LIN {X 0,Y 143.152,Z 440.148,A -85,B 0,C 180,E1 -24453.78,E2 -24453.78} C_VEL
LIN {X 0,Y 143.303,Z 440.124,A -85,B 0,C 180,E1 -24459.924,E2 -24459.924} C_VEL
LIN {X 0,Y 143.35,Z 440.119,A -85,B 0,C 180,E1 -24465.812,E2 -24465.812} C_VEL
LIN {X 0,Y 143.533,Z 440.103,A -85,B 0,C 180,E1 -24468.707,E2 -24468.707} C_VEL
LIN {X 0,Y 143.622,Z 440.089,A -85,B 0,C 180,E1 -24471.56,E2 -24471.56} C_VEL
LIN {X 0,Y 144.173,Z 439.992,A -85,B 0,C 180,E1 -24480.002,E2 -24480.002} C_VEL
LIN {X 0,Y 143.623,Z 440.096,A -85,B 0,C 180,E1 -24488.443,E2 -24488.443} C_VEL
LIN {X 0,Y 143.503,Z 440.112,A -85,B 0,C 180,E1 -24491.63,E2 -24491.63} C_VEL
LIN {X 0,Y 143.297,Z 440.142,A -85,B 0,C 180,E1 -24497.115,E2 -24497.115} C_VEL
LIN {X 0,Y 143.385,Z 440.981,A -85,B 0,C 180,E1 -24501.367,E2 -24501.367} C_VEL
LIN {X 0,Y 143.555,Z 442.59,A -85,B 0,C 180,E1 -24508.212,E2 -24508.212} C_VEL
LIN {X 0,Y 143.628,Z 443.352,A -85,B 0,C 180,E1 -24510.714,E2 -24510.714} C_VEL
LIN {X 0,Y 144.738,Z 446.525,A -85,B 0,C 180,E1 -24511.876,E2 -24511.876} C_VEL
LIN {X 0,Y 147.342,Z 449.815,A -85,B 0,C 180,E1 -24513.997,E2 -24513.997} C_VEL
LIN {X 0,Y 148.899,Z 453.219,A -85,B 0,C 180,E1 -24515.429,E2 -24515.429} C_VEL
LIN {X 0,Y 150.409,Z 455.407,A -85,B 0,C 180,E1 -24516.568,E2 -24516.568} C_VEL
LIN {X 0,Y 153.168,Z 461.405,A -85,B 0,C 180,E1 -24519.035,E2 -24519.035} C_VEL
LIN {X 0,Y 155.875,Z 468.036,A -85,B 0,C 180,E1 -24521.519,E2 -24521.519} C_VEL
LIN {X 0,Y 158.224,Z 476.972,A -85,B 0,C 180,E1 -24524.486,E2 -24524.486} C_VEL
LIN {X 0,Y 159.487,Z 487.574,A -85,B 0,C 180,E1 -24527.779,E2 -24527.779} C_VEL
LIN {X 0,Y 159.695,Z 496.347,A -85,B 0,C 180,E1 -24530.573,E2 -24530.573} C_VEL
LIN {X 0,Y 159.089,Z 505.794,A -85,B 0,C 180,E1 -24533.831,E2 -24533.831} C_VEL
LIN {X 0,Y 158.048,Z 512.286,A -85,B 0,C 180,E1 -24536.232,E2 -24536.232} C_VEL
LIN {X 0,Y 154.375,Z 520.117,A -85,B 0,C 180,E1 -24539.193,E2 -24539.193} C_VEL
LIN {X 0,Y 151.127,Z 526.657,A -85,B 0,C 180,E1 -24542.288,E2 -24542.288} C_VEL
LIN {X 0,Y 148.767,Z 531.159,A -85,B 0,C 180,E1 -24544.839,E2 -24544.839} C_VEL
LIN {X 0,Y 145.71,Z 536.651,A -85,B 0,C 180,E1 -24548.793,E2 -24548.793} C_VEL
LIN {X 0,Y 143.316,Z 540.978,A -85,B 0,C 180,E1 -24552.889,E2 -24552.889} C_VEL
LIN {X 0,Y 142.25,Z 543.351,A -85,B 0,C 180,E1 -24555.698,E2 -24555.698} C_VEL
LIN {X 0,Y 141.418,Z 545.156,A -85,B 0,C 180,E1 -24558.534,E2 -24558.534} C_VEL
LIN {X 0,Y 140.617,Z 547.617,A -85,B 0,C 180,E1 -24564.263,E2 -24564.263} C_VEL
LIN {X 0,Y 140.572,Z 548.37,A -85,B 0,C 180,E1 -24569.356,E2 -24569.356} C_VEL
LIN {X 0,Y 140.49,Z 548.211,A -85,B 0,C 180,E1 -24572.867,E2 -24572.867} C_VEL
LIN {X 0,Y 140.558,Z 547.615,A -85,B 0,C 180,E1 -24575.739,E2 -24575.739} C_VEL
LIN {X 0,Y 141.418,Z 545.156,A -85,B 0,C 180,E1 -24581.466,E2 -24581.466} C_VEL
LIN {X 0,Y 142.745,Z 542.198,A -85,B 0,C 180,E1 -24585.711,E2 -24585.711} C_VEL
LIN {X 0,Y 144.854,Z 538.206,A -85,B 0,C 180,E1 -24589.854,E2 -24589.854} C_VEL
LIN {X 0,Y 147.638,Z 533.074,A -85,B 0,C 180,E1 -24593.867,E2 -24593.867} C_VEL
LIN {X 0,Y 150.526,Z 527.813,A -85,B 0,C 180,E1 -24597.079,E2 -24597.079} C_VEL
LIN {X 0,Y 152.903,Z 523.006,A -85,B 0,C 180,E1 -24599.535,E2 -24599.535} C_VEL
LIN {X 0,Y 155.803,Z 517.169,A -85,B 0,C 180,E1 -24602.006,E2 -24602.006} C_VEL
LIN {X 0,Y 157.995,Z 512.284,A -85,B 0,C 180,E1 -24603.781,E2 -24603.781} C_VEL
LIN {X 0,Y 159.283,Z 504.165,A -85,B 0,C 180,E1 -24606.777,E2 -24606.777} C_VEL
LIN {X 0,Y 159.691,Z 494.189,A -85,B 0,C 180,E1 -24610.136,E2 -24610.136} C_VEL
LIN {X 0,Y 159.209,Z 484.217,A -85,B 0,C 180,E1 -24613.246,E2 -24613.246} C_VEL
LIN {X 0,Y 157.654,Z 474.494,A -85,B 0,C 180,E1 -24616.289,E2 -24616.289} C_VEL
LIN {X 0,Y 155.43,Z 466.702,A -85,B 0,C 180,E1 -24618.95,E2 -24618.95} C_VEL
LIN {X 0,Y 152.654,Z 459.906,A -85,B 0,C 180,E1 -24621.503,E2 -24621.503} C_VEL
LIN {X 0,Y 150.327,Z 455.158,A -85,B 0,C 180,E1 -24623.513,E2 -24623.513} C_VEL
LIN {X 0,Y 147.761,Z 451.088,A -85,B 0,C 180,E1 -24625.549,E2 -24625.549} C_VEL
LIN {X 0,Y 147.026,Z 449.221,A -85,B 0,C 180,E1 -24626.287,E2 -24626.287} C_VEL
LIN {X 0,Y 144.65,Z 446.353,A -85,B 0,C 180,E1 -24628.205,E2 -24628.205} C_VEL
LIN {X 0,Y 143.667,Z 443.599,A -85,B 0,C 180,E1 -24629.193,E2 -24629.193} C_VEL
LIN {X 0,Y 143.581,Z 443.188,A -85,B 0,C 180,E1 -24629.478,E2 -24629.478} C_VEL
LIN {X 0,Y 143.46,Z 442.211,A -85,B 0,C 180,E1 -24633.299,E2 -24633.299} C_VEL
LIN {X 0,Y 142.742,Z 441.762,A -85,B 0,C 180,E1 -24635.632,E2 -24635.632} C_VEL
LIN {X 0,Y 141.111,Z 441.498,A -85,B 0,C 180,E1 -24637.936,E2 -24637.936} C_VEL
LIN {X 0,Y 136.544,Z 441.058,A -85,B 0,C 180,E1 -24644.298,E2 -24644.298} C_VEL
LIN {X 0,Y 136.275,Z 441.006,A -85,B 0,C 180,E1 -24645.981,E2 -24645.981} C_VEL
LIN {X 0,Y 136.549,Z 440.977,A -85,B 0,C 180,E1 -24651.116,E2 -24651.116} C_VEL
LIN {X 0,Y 137.13,Z 440.867,A -85,B 0,C 180,E1 -24659.998,E2 -24659.998} C_VEL
LIN {X 0,Y 136.549,Z 440.967,A -85,B 0,C 180,E1 -24668.881,E2 -24668.881} C_VEL
LIN {X 0,Y 136.437,Z 440.991,A -85,B 0,C 180,E1 -24671.889,E2 -24671.889} C_VEL
LIN {X 0,Y 136.235,Z 441.013,A -85,B 0,C 180,E1 -24678.029,E2 -24678.029} C_VEL
LIN {X 0,Y 136.194,Z 441.018,A -85,B 0,C 180,E1 -24681.747,E2 -24681.747} C_VEL
LIN {X 0,Y 136.08,Z 441.049,A -85,B 0,C 180,E1 -24685.115,E2 -24685.115} C_VEL
LIN {X 0,Y 136.755,Z 443.236,A -85,B 0,C 180,E1 -24686.104,E2 -24686.104} C_VEL
LIN {X 0,Y 138.766,Z 445.73,A -85,B 0,C 180,E1 -24688.327,E2 -24688.327} C_VEL
LIN {X 0,Y 140.093,Z 446.714,A -85,B 0,C 180,E1 -24689.543,E2 -24689.543} C_VEL
LIN {X 0,Y 141.491,Z 449.595,A -85,B 0,C 180,E1 -24691.122,E2 -24691.122} C_VEL
LIN {X 0,Y 143.665,Z 452.032,A -85,B 0,C 180,E1 -24693.012,E2 -24693.012} C_VEL
LIN {X 0,Y 145.332,Z 454.972,A -85,B 0,C 180,E1 -24694.707,E2 -24694.707} C_VEL
LIN {X 0,Y 148.827,Z 460.554,A -85,B 0,C 180,E1 -24697.87,E2 -24697.87} C_VEL
LIN {X 0,Y 153.54,Z 470.176,A -85,B 0,C 180,E1 -24702.464,E2 -24702.464} C_VEL
LIN {X 0,Y 157.143,Z 479.374,A -85,B 0,C 180,E1 -24706.461,E2 -24706.461} C_VEL
LIN {X 0,Y 159.474,Z 487.535,A -85,B 0,C 180,E1 -24709.834,E2 -24709.834} C_VEL
LIN {X 0,Y 161.218,Z 496.736,A -85,B 0,C 180,E1 -24713.624,E2 -24713.624} C_VEL
LIN {X 0,Y 162.342,Z 505.111,A -85,B 0,C 180,E1 -24717.36,E2 -24717.36} C_VEL
LIN {X 0,Y 164.436,Z 512.684,A -85,B 0,C 180,E1 -24721.389,E2 -24721.389} C_VEL
LIN {X 0,Y 167.413,Z 518.734,A -85,B 0,C 180,E1 -24725.179,E2 -24725.179} C_VEL
LIN {X 0,Y 170.704,Z 523.029,A -85,B 0,C 180,E1 -24728.252,E2 -24728.252} C_VEL
LIN {X 0,Y 176.708,Z 528.218,A -85,B 0,C 180,E1 -24732.649,E2 -24732.649} C_VEL
LIN {X 0,Y 183.955,Z 532.227,A -85,B 0,C 180,E1 -24736.749,E2 -24736.749} C_VEL
LIN {X 0,Y 192.338,Z 535.226,A -85,B 0,C 180,E1 -24740.593,E2 -24740.593} C_VEL
LIN {X 0,Y 200.865,Z 537.166,A -85,B 0,C 180,E1 -24743.975,E2 -24743.975} C_VEL
LIN {X 0,Y 206.622,Z 538.036,A -85,B 0,C 180,E1 -24746.099,E2 -24746.099} C_VEL
LIN {X 0,Y 212.047,Z 538.453,A -85,B 0,C 180,E1 -24748.101,E2 -24748.101} C_VEL
LIN {X 0,Y 216.311,Z 538.505,A -85,B 0,C 180,E1 -24750,E2 -24750} C_VEL
LIN {X 0,Y 211.001,Z 538.385,A -85,B 0,C 180,E1 -24752.268,E2 -24752.268} C_VEL
LIN {X 0,Y 204.489,Z 537.779,A -85,B 0,C 180,E1 -24754.678,E2 -24754.678} C_VEL
LIN {X 0,Y 195.02,Z 535.982,A -85,B 0,C 180,E1 -24758.288,E2 -24758.288} C_VEL
LIN {X 0,Y 186.734,Z 533.39,A -85,B 0,C 180,E1 -24761.896,E2 -24761.896} C_VEL
LIN {X 0,Y 178.979,Z 529.663,A -85,B 0,C 180,E1 -24765.954,E2 -24765.954} C_VEL
LIN {X 0,Y 174.564,Z 526.656,A -85,B 0,C 180,E1 -24768.788,E2 -24768.788} C_VEL
LIN {X 0,Y 169.225,Z 521.23,A -85,B 0,C 180,E1 -24773.069,E2 -24773.069} C_VEL
LIN {X 0,Y 165.611,Z 515.406,A -85,B 0,C 180,E1 -24776.982,E2 -24776.982} C_VEL
LIN {X 0,Y 163.318,Z 509.057,A -85,B 0,C 180,E1 -24780.613,E2 -24780.613} C_VEL
LIN {X 0,Y 162.063,Z 503.157,A -85,B 0,C 180,E1 -24783.563,E2 -24783.563} C_VEL
LIN {X 0,Y 160.944,Z 494.761,A -85,B 0,C 180,E1 -24787.167,E2 -24787.167} C_VEL
LIN {X 0,Y 159.114,Z 486.266,A -85,B 0,C 180,E1 -24790.677,E2 -24790.677} C_VEL
LIN {X 0,Y 156.632,Z 477.951,A -85,B 0,C 180,E1 -24794.12,E2 -24794.12} C_VEL
LIN {X 0,Y 152.851,Z 468.714,A -85,B 0,C 180,E1 -24798.189,E2 -24798.189} C_VEL
LIN {X 0,Y 148.798,Z 460.661,A -85,B 0,C 180,E1 -24802.122,E2 -24802.122} C_VEL
LIN {X 0,Y 145.994,Z 455.806,A -85,B 0,C 180,E1 -24804.715,E2 -24804.715} C_VEL
LIN {X 0,Y 143.909,Z 452.642,A -85,B 0,C 180,E1 -24806.707,E2 -24806.707} C_VEL
LIN {X 0,Y 143.083,Z 451.254,A -85,B 0,C 180,E1 -24807.506,E2 -24807.506} C_VEL
LIN {X 0,Y 140.829,Z 448.546,A -85,B 0,C 180,E1 -24809.548,E2 -24809.548} C_VEL
LIN {X 0,Y 139.946,Z 446.499,A -85,B 0,C 180,E1 -24810.611,E2 -24810.611} C_VEL
LIN {X 0,Y 137.323,Z 444.183,A -85,B 0,C 180,E1 -24813.193,E2 -24813.193} C_VEL
LIN {X 0,Y 136.247,Z 441.855,A -85,B 0,C 180,E1 -24814.612,E2 -24814.612} C_VEL
LIN {X 0,Y 136.079,Z 441.024,A -85,B 0,C 180,E1 -24814.987,E2 -24814.987} C_VEL
LIN {X 0,Y 136.239,Z 441.008,A -85,B 0,C 180,E1 -24818.834,E2 -24818.834} C_VEL
LIN {X 0,Y 136.26,Z 441.001,A -85,B 0,C 180,E1 -24825.057,E2 -24825.057} C_VEL
LIN {X 0,Y 136.428,Z 440.991,A -85,B 0,C 180,E1 -24828.167,E2 -24828.167} C_VEL
LIN {X 0,Y 136.548,Z 440.967,A -85,B 0,C 180,E1 -24831.119,E2 -24831.119} C_VEL
LIN {X 0,Y 137.13,Z 440.867,A -85,B 0,C 180,E1 -24840.002,E2 -24840.002} C_VEL
LIN {X 0,Y 136.549,Z 440.976,A -85,B 0,C 180,E1 -24848.884,E2 -24848.884} C_VEL
LIN {X 0,Y 136.439,Z 440.993,A -85,B 0,C 180,E1 -24851.892,E2 -24851.892} C_VEL
LIN {X 0,Y 136.262,Z 441.014,A -85,B 0,C 180,E1 -24854.946,E2 -24854.946} C_VEL
LIN {X 0,Y 136.364,Z 442.037,A -85,B 0,C 180,E1 -24861.149,E2 -24861.149} C_VEL
LIN {X 0,Y 136.444,Z 443.198,A -85,B 0,C 180,E1 -24865.251,E2 -24865.251} C_VEL
LIN {X 0,Y 137.466,Z 445.953,A -85,B 0,C 180,E1 -24866.575,E2 -24866.575} C_VEL
LIN {X 0,Y 139.977,Z 449.017,A -85,B 0,C 180,E1 -24869.142,E2 -24869.142} C_VEL
LIN {X 0,Y 140.494,Z 449.746,A -85,B 0,C 180,E1 -24869.662,E2 -24869.662} C_VEL
LIN {X 0,Y 142.053,Z 453.203,A -85,B 0,C 180,E1 -24871.403,E2 -24871.403} C_VEL
LIN {X 0,Y 143.833,Z 455.627,A -85,B 0,C 180,E1 -24872.972,E2 -24872.972} C_VEL
LIN {X 0,Y 145.746,Z 459.585,A -85,B 0,C 180,E1 -24874.942,E2 -24874.942} C_VEL
LIN {X 0,Y 149.295,Z 467.386,A -85,B 0,C 180,E1 -24878.488,E2 -24878.488} C_VEL
LIN {X 0,Y 151.713,Z 475.064,A -85,B 0,C 180,E1 -24881.511,E2 -24881.511} C_VEL
LIN {X 0,Y 152.981,Z 482.109,A -85,B 0,C 180,E1 -24883.986,E2 -24883.986} C_VEL
LIN {X 0,Y 153.608,Z 490.094,A -85,B 0,C 180,E1 -24886.664,E2 -24886.664} C_VEL
LIN {X 0,Y 153.606,Z 496.767,A -85,B 0,C 180,E1 -24888.922,E2 -24888.922} C_VEL
LIN {X 0,Y 153.015,Z 505.059,A -85,B 0,C 180,E1 -24891.926,E2 -24891.926} C_VEL
LIN {X 0,Y 151.949,Z 512.081,A -85,B 0,C 180,E1 -24894.68,E2 -24894.68} C_VEL
LIN {X 0,Y 150.668,Z 515.347,A -85,B 0,C 180,E1 -24895.963,E2 -24895.963} C_VEL
LIN {X 0,Y 147.535,Z 521.295,A -85,B 0,C 180,E1 -24898.4,E2 -24898.4} C_VEL
LIN {X 0,Y 144.83,Z 526.459,A -85,B 0,C 180,E1 -24900.971,E2 -24900.971} C_VEL
LIN {X 0,Y 142.372,Z 530.962,A -85,B 0,C 180,E1 -24903.624,E2 -24903.624} C_VEL
LIN {X 0,Y 139.088,Z 536.453,A -85,B 0,C 180,E1 -24907.731,E2 -24907.731} C_VEL
LIN {X 0,Y 136.51,Z 540.78,A -85,B 0,C 180,E1 -24912.007,E2 -24912.007} C_VEL
LIN {X 0,Y 135.352,Z 543.153,A -85,B 0,C 180,E1 -24914.953,E2 -24914.953} C_VEL
LIN {X 0,Y 134.452,Z 544.958,A -85,B 0,C 180,E1 -24917.932,E2 -24917.932} C_VEL
LIN {X 0,Y 133.543,Z 547.419,A -85,B 0,C 180,E1 -24923.958,E2 -24923.958} C_VEL
LIN {X 0,Y 133.414,Z 548.014,A -85,B 0,C 180,E1 -24926.98,E2 -24926.98} C_VEL
LIN {X 0,Y 133.536,Z 548.175,A -85,B 0,C 180,E1 -24930,E2 -24930} C_VEL
LIN {X 0,Y 133.401,Z 548.014,A -85,B 0,C 180,E1 -24933.02,E2 -24933.02} C_VEL
LIN {X 0,Y 133.474,Z 547.417,A -85,B 0,C 180,E1 -24936.045,E2 -24936.045} C_VEL
LIN {X 0,Y 134.452,Z 544.958,A -85,B 0,C 180,E1 -24942.068,E2 -24942.068} C_VEL
LIN {X 0,Y 135.884,Z 542,A -85,B 0,C 180,E1 -24946.526,E2 -24946.526} C_VEL
LIN {X 0,Y 138.16,Z 538.008,A -85,B 0,C 180,E1 -24950.859,E2 -24950.859} C_VEL
LIN {X 0,Y 141.152,Z 532.876,A -85,B 0,C 180,E1 -24955.037,E2 -24955.037} C_VEL
LIN {X 0,Y 143.618,Z 528.772,A -85,B 0,C 180,E1 -24957.702,E2 -24957.702} C_VEL
LIN {X 0,Y 146.723,Z 522.808,A -85,B 0,C 180,E1 -24960.912,E2 -24960.912} C_VEL
LIN {X 0,Y 149.807,Z 516.971,A -85,B 0,C 180,E1 -24963.451,E2 -24963.451} C_VEL
LIN {X 0,Y 151.364,Z 513.716,A -85,B 0,C 180,E1 -24964.664,E2 -24964.664} C_VEL
LIN {X 0,Y 152.584,Z 508.373,A -85,B 0,C 180,E1 -24966.782,E2 -24966.782} C_VEL
LIN {X 0,Y 153.37,Z 501.695,A -85,B 0,C 180,E1 -24969.313,E2 -24969.313} C_VEL
LIN {X 0,Y 153.667,Z 493.139,A -85,B 0,C 180,E1 -24972.324,E2 -24972.324} C_VEL
LIN {X 0,Y 153.368,Z 485.551,A -85,B 0,C 180,E1 -24974.895,E2 -24974.895} C_VEL
LIN {X 0,Y 152.082,Z 476.72,A -85,B 0,C 180,E1 -24977.924,E2 -24977.924} C_VEL
LIN {X 0,Y 149.999,Z 469.293,A -85,B 0,C 180,E1 -24980.692,E2 -24980.692} C_VEL
LIN {X 0,Y 147.381,Z 463.041,A -85,B 0,C 180,E1 -24983.409,E2 -24983.409} C_VEL
LIN {X 0,Y 145.755,Z 459.586,A -85,B 0,C 180,E1 -24985.053,E2 -24985.053} C_VEL
LIN {X 0,Y 143.834,Z 455.622,A -85,B 0,C 180,E1 -24987.028,E2 -24987.028} C_VEL
LIN {X 0,Y 140.918,Z 451.084,A -85,B 0,C 180,E1 -24989.773,E2 -24989.773} C_VEL
LIN {X 0,Y 140.363,Z 449.264,A -85,B 0,C 180,E1 -24990.53,E2 -24990.53} C_VEL
LIN {X 0,Y 137.692,Z 446.36,A -85,B 0,C 180,E1 -24993.165,E2 -24993.165} C_VEL
LIN {X 0,Y 136.48,Z 443.495,A -85,B 0,C 180,E1 -24994.654,E2 -24994.654} C_VEL
LIN {X 0,Y 136.387,Z 442.867,A -85,B 0,C 180,E1 -24994.942,E2 -24994.942} C_VEL
LIN {X 0,Y 136.363,Z 442.035,A -85,B 0,C 180,E1 -24998.851,E2 -24998.851} C_VEL
LIN {X 0,Y 136.262,Z 441.012,A -85,B 0,C 180,E1 -25005.054,E2 -25005.054} C_VEL
LIN {X 0,Y 136.275,Z 441.006,A -85,B 0,C 180,E1 -25005.981,E2 -25005.981} C_VEL
LIN {X 0,Y 135.666,Z 441.087,A -85,B 0,C 180,E1 -25008.449,E2 -25008.449} C_VEL
LIN {X 0,Y 134.131,Z 441.278,A -85,B 0,C 180,E1 -25010.888,E2 -25010.888} C_VEL
LIN {X 0,Y 130.654,Z 441.709,A -85,B 0,C 180,E1 -25015.879,E2 -25015.879} C_VEL
LIN {X 0,Y 129.914,Z 441.783,A -85,B 0,C 180,E1 -25018.501,E2 -25018.501} C_VEL
LIN {X 0,Y 129.972,Z 441.761,A -85,B 0,C 180,E1 -25019.384,E2 -25019.384} C_VEL
LIN {X 0,Y 130.085,Z 441.743,A -85,B 0,C 180,E1 -25019.998,E2 -25019.998} C_VEL
LIN {X 0,Y 129.472,Z 441.847,A -85,B 0,C 180,E1 -25029.37,E2 -25029.37} C_VEL
LIN {X 0,Y 129.341,Z 441.874,A -85,B 0,C 180,E1 -25032.552,E2 -25032.552} C_VEL
LIN {X 0,Y 129.192,Z 442.042,A -85,B 0,C 180,E1 -25037.612,E2 -25037.612} C_VEL
LIN {X 0,Y 129.975,Z 444.408,A -85,B 0,C 180,E1 -25039.339,E2 -25039.339} C_VEL
LIN {X 0,Y 132.566,Z 447.181,A -85,B 0,C 180,E1 -25043.163,E2 -25043.163} C_VEL
LIN {X 0,Y 133.355,Z 447.728,A -85,B 0,C 180,E1 -25044.105,E2 -25044.105} C_VEL
LIN {X 0,Y 134.792,Z 450.708,A -85,B 0,C 180,E1 -25046.201,E2 -25046.201} C_VEL
LIN {X 0,Y 137.341,Z 453.815,A -85,B 0,C 180,E1 -25049.087,E2 -25049.087} C_VEL
LIN {X 0,Y 138.451,Z 455.857,A -85,B 0,C 180,E1 -25050.503,E2 -25050.503} C_VEL
LIN {X 0,Y 139.798,Z 457.375,A -85,B 0,C 180,E1 -25051.859,E2 -25051.859} C_VEL
LIN {X 0,Y 143.013,Z 463.032,A -85,B 0,C 180,E1 -25055.353,E2 -25055.353} C_VEL
LIN {X 0,Y 146.78,Z 470.562,A -85,B 0,C 180,E1 -25059.522,E2 -25059.522} C_VEL
LIN {X 0,Y 150.046,Z 478.638,A -85,B 0,C 180,E1 -25063.518,E2 -25063.518} C_VEL
LIN {X 0,Y 152.68,Z 487.147,A -85,B 0,C 180,E1 -25067.431,E2 -25067.431} C_VEL
LIN {X 0,Y 154.244,Z 494.584,A -85,B 0,C 180,E1 -25070.766,E2 -25070.766} C_VEL
LIN {X 0,Y 155.145,Z 501.503,A -85,B 0,C 180,E1 -25073.922,E2 -25073.922} C_VEL
LIN {X 0,Y 156.187,Z 509.493,A -85,B 0,C 180,E1 -25077.924,E2 -25077.924} C_VEL
LIN {X 0,Y 158.536,Z 516.995,A -85,B 0,C 180,E1 -25082.448,E2 -25082.448} C_VEL
LIN {X 0,Y 162.311,Z 523.278,A -85,B 0,C 180,E1 -25087.065,E2 -25087.065} C_VEL
LIN {X 0,Y 167.764,Z 528.419,A -85,B 0,C 180,E1 -25091.646,E2 -25091.646} C_VEL
LIN {X 0,Y 174.661,Z 532.488,A -85,B 0,C 180,E1 -25096.03,E2 -25096.03} C_VEL
LIN {X 0,Y 179.811,Z 534.632,A -85,B 0,C 180,E1 -25098.731,E2 -25098.731} C_VEL
LIN {X 0,Y 185.399,Z 536.246,A -85,B 0,C 180,E1 -25101.279,E2 -25101.279} C_VEL
LIN {X 0,Y 197.271,Z 538.308,A -85,B 0,C 180,E1 -25105.955,E2 -25105.955} C_VEL
LIN {X 0,Y 203.89,Z 538.764,A -85,B 0,C 180,E1 -25108.373,E2 -25108.373} C_VEL
LIN {X 0,Y 207.943,Z 538.733,A -85,B 0,C 180,E1 -25110,E2 -25110} C_VEL
LIN {X 0,Y 202.902,Z 538.706,A -85,B 0,C 180,E1 -25111.985,E2 -25111.985} C_VEL
LIN {X 0,Y 197.148,Z 538.298,A -85,B 0,C 180,E1 -25114.088,E2 -25114.088} C_VEL
LIN {X 0,Y 184.954,Z 536.128,A -85,B 0,C 180,E1 -25118.906,E2 -25118.906} C_VEL
LIN {X 0,Y 179.306,Z 534.463,A -85,B 0,C 180,E1 -25121.518,E2 -25121.518} C_VEL
LIN {X 0,Y 172.174,Z 531.319,A -85,B 0,C 180,E1 -25125.401,E2 -25125.401} C_VEL
LIN {X 0,Y 165.053,Z 526.107,A -85,B 0,C 180,E1 -25130.489,E2 -25130.489} C_VEL
LIN {X 0,Y 160.65,Z 520.863,A -85,B 0,C 180,E1 -25134.757,E2 -25134.757} C_VEL
LIN {X 0,Y 157.739,Z 515.011,A -85,B 0,C 180,E1 -25138.792,E2 -25138.792} C_VEL
LIN {X 0,Y 155.969,Z 508.24,A -85,B 0,C 180,E1 -25142.732,E2 -25142.732} C_VEL
LIN {X 0,Y 155.167,Z 501.502,A -85,B 0,C 180,E1 -25146.072,E2 -25146.072} C_VEL
LIN {X 0,Y 154.242,Z 494.588,A -85,B 0,C 180,E1 -25149.234,E2 -25149.234} C_VEL
LIN {X 0,Y 152.679,Z 487.149,A -85,B 0,C 180,E1 -25152.568,E2 -25152.568} C_VEL
LIN {X 0,Y 150.029,Z 478.61,A -85,B 0,C 180,E1 -25156.498,E2 -25156.498} C_VEL
LIN {X 0,Y 146.751,Z 470.581,A -85,B 0,C 180,E1 -25160.486,E2 -25160.486} C_VEL
LIN {X 0,Y 142.215,Z 461.47,A -85,B 0,C 180,E1 -25165.551,E2 -25165.551} C_VEL
LIN {X 0,Y 140.368,Z 458.597,A -85,B 0,C 180,E1 -25167.438,E2 -25167.438} C_VEL
LIN {X 0,Y 139.797,Z 457.38,A -85,B 0,C 180,E1 -25168.141,E2 -25168.141} C_VEL
LIN {X 0,Y 138.121,Z 455.345,A -85,B 0,C 180,E1 -25169.882,E2 -25169.882} C_VEL
LIN {X 0,Y 136.142,Z 452.123,A -85,B 0,C 180,E1 -25172.317,E2 -25172.317} C_VEL
LIN {X 0,Y 133.974,Z 449.353,A -85,B 0,C 180,E1 -25174.878,E2 -25174.878} C_VEL
LIN {X 0,Y 133.227,Z 447.52,A -85,B 0,C 180,E1 -25176.077,E2 -25176.077} C_VEL
LIN {X 0,Y 130.715,Z 445.463,A -85,B 0,C 180,E1 -25179.397,E2 -25179.397} C_VEL
LIN {X 0,Y 129.515,Z 443.301,A -85,B 0,C 180,E1 -25181.616,E2 -25181.616} C_VEL
LIN {X 0,Y 129.19,Z 441.893,A -85,B 0,C 180,E1 -25182.592,E2 -25182.592} C_VEL
LIN {X 0,Y 129.373,Z 441.87,A -85,B 0,C 180,E1 -25187.905,E2 -25187.905} C_VEL
LIN {X 0,Y 129.471,Z 441.847,A -85,B 0,C 180,E1 -25190.63,E2 -25190.63} C_VEL
LIN {X 0,Y 130.085,Z 441.743,A -85,B 0,C 180,E1 -25200.002,E2 -25200.002} C_VEL
LIN {X 0,Y 129.472,Z 441.858,A -85,B 0,C 180,E1 -25209.374,E2 -25209.374} C_VEL
LIN {X 0,Y 129.342,Z 441.876,A -85,B 0,C 180,E1 -25212.555,E2 -25212.555} C_VEL
LIN {X 0,Y 129.261,Z 442.629,A -85,B 0,C 180,E1 -25217.3,E2 -25217.3} C_VEL
LIN {X 0,Y 130.424,Z 445.76,A -85,B 0,C 180,E1 -25219.58,E2 -25219.58} C_VEL
LIN {X 0,Y 133.372,Z 449.115,A -85,B 0,C 180,E1 -25223.692,E2 -25223.692} C_VEL
LIN {X 0,Y 133.814,Z 449.957,A -85,B 0,C 180,E1 -25224.33,E2 -25224.33} C_VEL
LIN {X 0,Y 135.361,Z 453.257,A -85,B 0,C 180,E1 -25226.501,E2 -25226.501} C_VEL
LIN {X 0,Y 137.281,Z 455.719,A -85,B 0,C 180,E1 -25228.579,E2 -25228.579} C_VEL
LIN {X 0,Y 138.82,Z 459.231,A -85,B 0,C 180,E1 -25230.612,E2 -25230.612} C_VEL
LIN {X 0,Y 139.967,Z 460.897,A -85,B 0,C 180,E1 -25231.818,E2 -25231.818} C_VEL
LIN {X 0,Y 143.496,Z 468.921,A -85,B 0,C 180,E1 -25235.997,E2 -25235.997} C_VEL
LIN {X 0,Y 145.958,Z 476.275,A -85,B 0,C 180,E1 -25239.287,E2 -25239.287} C_VEL
LIN {X 0,Y 147.347,Z 484.091,A -85,B 0,C 180,E1 -25242.349,E2 -25242.349} C_VEL
LIN {X 0,Y 147.789,Z 492.75,A -85,B 0,C 180,E1 -25245.507,E2 -25245.507} C_VEL
LIN {X 0,Y 147.255,Z 503.201,A -85,B 0,C 180,E1 -25249.404,E2 -25249.404} C_VEL
LIN {X 0,Y 145.888,Z 511.872,A -85,B 0,C 180,E1 -25252.975,E2 -25252.975} C_VEL
LIN {X 0,Y 144.799,Z 515.148,A -85,B 0,C 180,E1 -25254.379,E2 -25254.379} C_VEL
LIN {X 0,Y 141.515,Z 521.097,A -85,B 0,C 180,E1 -25256.888,E2 -25256.888} C_VEL
LIN {X 0,Y 137.991,Z 527.352,A -85,B 0,C 180,E1 -25260.18,E2 -25260.18} C_VEL
LIN {X 0,Y 136.047,Z 530.765,A -85,B 0,C 180,E1 -25262.295,E2 -25262.295} C_VEL
LIN {X 0,Y 132.519,Z 536.255,A -85,B 0,C 180,E1 -25266.563,E2 -25266.563} C_VEL
LIN {X 0,Y 129.742,Z 540.581,A -85,B 0,C 180,E1 -25271.034,E2 -25271.034} C_VEL
LIN {X 0,Y 128.466,Z 542.955,A -85,B 0,C 180,E1 -25274.126,E2 -25274.126} C_VEL
LIN {X 0,Y 127.481,Z 544.76,A -85,B 0,C 180,E1 -25277.261,E2 -25277.261} C_VEL
LIN {X 0,Y 126.464,Z 547.222,A -85,B 0,C 180,E1 -25283.619,E2 -25283.619} C_VEL
LIN {X 0,Y 126.317,Z 547.817,A -85,B 0,C 180,E1 -25286.811,E2 -25286.811} C_VEL
LIN {X 0,Y 126.432,Z 547.978,A -85,B 0,C 180,E1 -25290,E2 -25290} C_VEL
LIN {X 0,Y 126.306,Z 547.817,A -85,B 0,C 180,E1 -25293.19,E2 -25293.19} C_VEL
LIN {X 0,Y 126.415,Z 547.22,A -85,B 0,C 180,E1 -25296.384,E2 -25296.384} C_VEL
LIN {X 0,Y 127.481,Z 544.76,A -85,B 0,C 180,E1 -25302.739,E2 -25302.739} C_VEL
LIN {X 0,Y 129.062,Z 541.802,A -85,B 0,C 180,E1 -25307.427,E2 -25307.427} C_VEL
LIN {X 0,Y 131.521,Z 537.81,A -85,B 0,C 180,E1 -25311.965,E2 -25311.965} C_VEL
LIN {X 0,Y 134.739,Z 532.679,A -85,B 0,C 180,E1 -25316.318,E2 -25316.318} C_VEL
LIN {X 0,Y 137.24,Z 528.729,A -85,B 0,C 180,E1 -25318.997,E2 -25318.997} C_VEL
LIN {X 0,Y 140.724,Z 522.472,A -85,B 0,C 180,E1 -25322.47,E2 -25322.47} C_VEL
LIN {X 0,Y 143.923,Z 516.774,A -85,B 0,C 180,E1 -25325.013,E2 -25325.013} C_VEL
LIN {X 0,Y 145.41,Z 513.513,A -85,B 0,C 180,E1 -25326.303,E2 -25326.303} C_VEL
LIN {X 0,Y 146.691,Z 507.118,A -85,B 0,C 180,E1 -25328.995,E2 -25328.995} C_VEL
LIN {X 0,Y 147.49,Z 499.878,A -85,B 0,C 180,E1 -25331.843,E2 -25331.843} C_VEL
LIN {X 0,Y 147.766,Z 491.738,A -85,B 0,C 180,E1 -25334.854,E2 -25334.854} C_VEL
LIN {X 0,Y 147.176,Z 483.046,A -85,B 0,C 180,E1 -25338.044,E2 -25338.044} C_VEL
LIN {X 0,Y 145.656,Z 475.203,A -85,B 0,C 180,E1 -25341.15,E2 -25341.15} C_VEL
LIN {X 0,Y 143.223,Z 468.266,A -85,B 0,C 180,E1 -25344.342,E2 -25344.342} C_VEL
LIN {X 0,Y 139.967,Z 460.897,A -85,B 0,C 180,E1 -25348.182,E2 -25348.182} C_VEL
LIN {X 0,Y 138.11,Z 457.89,A -85,B 0,C 180,E1 -25350.253,E2 -25350.253} C_VEL
LIN {X 0,Y 136.907,Z 455.025,A -85,B 0,C 180,E1 -25351.858,E2 -25351.858} C_VEL
LIN {X 0,Y 134.509,Z 451.848,A -85,B 0,C 180,E1 -25354.567,E2 -25354.567} C_VEL
LIN {X 0,Y 133.549,Z 449.128,A -85,B 0,C 180,E1 -25356.135,E2 -25356.135} C_VEL
LIN {X 0,Y 130.828,Z 446.386,A -85,B 0,C 180,E1 -25359.766,E2 -25359.766} C_VEL
LIN {X 0,Y 129.548,Z 443.693,A -85,B 0,C 180,E1 -25362.027,E2 -25362.027} C_VEL
LIN {X 0,Y 129.228,Z 442.439,A -85,B 0,C 180,E1 -25362.798,E2 -25362.798} C_VEL
LIN {X 0,Y 129.374,Z 441.87,A -85,B 0,C 180,E1 -25367.902,E2 -25367.902} C_VEL
LIN {X 0,Y 129.472,Z 441.858,A -85,B 0,C 180,E1 -25370.626,E2 -25370.626} C_VEL
LIN {X 0,Y 129.972,Z 441.761,A -85,B 0,C 180,E1 -25379.384,E2 -25379.384} C_VEL
LIN {X 0,Y 129.903,Z 441.912,A -85,B 0,C 180,E1 -25381.102,E2 -25381.102} C_VEL
LIN {X 0,Y 128.827,Z 442.724,A -85,B 0,C 180,E1 -25383.643,E2 -25383.643} C_VEL
LIN {X 0,Y 125.305,Z 445.94,A -85,B 0,C 180,E1 -25389.61,E2 -25389.61} C_VEL
LIN {X 0,Y 124.974,Z 447.305,A -85,B 0,C 180,E1 -25392.287,E2 -25392.287} C_VEL
LIN {X 0,Y 125.216,Z 447.687,A -85,B 0,C 180,E1 -25393.181,E2 -25393.181} C_VEL
LIN {X 0,Y 126.971,Z 448.884,A -85,B 0,C 180,E1 -25396.788,E2 -25396.788} C_VEL
LIN {X 0,Y 127.806,Z 451.163,A -85,B 0,C 180,E1 -25398.846,E2 -25398.846} C_VEL
LIN {X 0,Y 130.676,Z 454.297,A -85,B 0,C 180,E1 -25403.323,E2 -25403.323} C_VEL
LIN {X 0,Y 131.731,Z 456.709,A -85,B 0,C 180,E1 -25405.263,E2 -25405.263} C_VEL
LIN {X 0,Y 133.934,Z 459.653,A -85,B 0,C 180,E1 -25408.179,E2 -25408.179} C_VEL
LIN {X 0,Y 135.124,Z 461.883,A -85,B 0,C 180,E1 -25409.797,E2 -25409.797} C_VEL
LIN {X 0,Y 136.223,Z 463.251,A -85,B 0,C 180,E1 -25411.057,E2 -25411.057} C_VEL
LIN {X 0,Y 140.118,Z 470.912,A -85,B 0,C 180,E1 -25416.109,E2 -25416.109} C_VEL
LIN {X 0,Y 143.362,Z 478.793,A -85,B 0,C 180,E1 -25420.586,E2 -25420.586} C_VEL
LIN {X 0,Y 145.712,Z 486.1,A -85,B 0,C 180,E1 -25424.372,E2 -25424.372} C_VEL
LIN {X 0,Y 147.526,Z 493.778,A -85,B 0,C 180,E1 -25428.169,E2 -25428.169} C_VEL
LIN {X 0,Y 148.488,Z 500.347,A -85,B 0,C 180,E1 -25431.389,E2 -25431.389} C_VEL
LIN {X 0,Y 148.994,Z 507.266,A -85,B 0,C 180,E1 -25434.901,E2 -25434.901} C_VEL
LIN {X 0,Y 149.869,Z 513.33,A -85,B 0,C 180,E1 -25438.411,E2 -25438.411} C_VEL
LIN {X 0,Y 151.782,Z 519.211,A -85,B 0,C 180,E1 -25442.418,E2 -25442.418} C_VEL
LIN {X 0,Y 154.175,Z 523.521,A -85,B 0,C 180,E1 -25445.779,E2 -25445.779} C_VEL
LIN {X 0,Y 159.241,Z 528.868,A -85,B 0,C 180,E1 -25450.806,E2 -25450.806} C_VEL
LIN {X 0,Y 165.393,Z 532.748,A -85,B 0,C 180,E1 -25455.229,E2 -25455.229} C_VEL
LIN {X 0,Y 171.882,Z 535.382,A -85,B 0,C 180,E1 -25458.902,E2 -25458.902} C_VEL
LIN {X 0,Y 177.591,Z 536.978,A -85,B 0,C 180,E1 -25461.621,E2 -25461.621} C_VEL
LIN {X 0,Y 187.526,Z 538.563,A -85,B 0,C 180,E1 -25465.701,E2 -25465.701} C_VEL
LIN {X 0,Y 196.804,Z 539.034,A -85,B 0,C 180,E1 -25469.089,E2 -25469.089} C_VEL
LIN {X 0,Y 199.217,Z 538.97,A -85,B 0,C 180,E1 -25470,E2 -25470} C_VEL
LIN {X 0,Y 193.549,Z 538.964,A -85,B 0,C 180,E1 -25472.081,E2 -25472.081} C_VEL
LIN {X 0,Y 183.663,Z 538.054,A -85,B 0,C 180,E1 -25475.798,E2 -25475.798} C_VEL
LIN {X 0,Y 175.773,Z 536.512,A -85,B 0,C 180,E1 -25479.203,E2 -25479.203} C_VEL
LIN {X 0,Y 170.374,Z 534.899,A -85,B 0,C 180,E1 -25481.903,E2 -25481.903} C_VEL
LIN {X 0,Y 161.842,Z 530.737,A -85,B 0,C 180,E1 -25487.192,E2 -25487.192} C_VEL
LIN {X 0,Y 157.335,Z 527.157,A -85,B 0,C 180,E1 -25490.937,E2 -25490.937} C_VEL
LIN {X 0,Y 152.937,Z 521.428,A -85,B 0,C 180,E1 -25495.882,E2 -25495.882} C_VEL
LIN {X 0,Y 150.5,Z 515.567,A -85,B 0,C 180,E1 -25500.131,E2 -25500.131} C_VEL
LIN {X 0,Y 149.284,Z 509.768,A -85,B 0,C 180,E1 -25503.728,E2 -25503.728} C_VEL
LIN {X 0,Y 148.645,Z 501.728,A -85,B 0,C 180,E1 -25507.925,E2 -25507.925} C_VEL
LIN {X 0,Y 147.693,Z 494.961,A -85,B 0,C 180,E1 -25511.285,E2 -25511.285} C_VEL
LIN {X 0,Y 146.175,Z 487.728,A -85,B 0,C 180,E1 -25514.836,E2 -25514.836} C_VEL
LIN {X 0,Y 143.966,Z 480.609,A -85,B 0,C 180,E1 -25518.505,E2 -25518.505} C_VEL
LIN {X 0,Y 140.635,Z 472.229,A -85,B 0,C 180,E1 -25523.155,E2 -25523.155} C_VEL
LIN {X 0,Y 137.801,Z 466.425,A -85,B 0,C 180,E1 -25526.754,E2 -25526.754} C_VEL
LIN {X 0,Y 136.218,Z 463.262,A -85,B 0,C 180,E1 -25528.942,E2 -25528.942} C_VEL
LIN {X 0,Y 134.501,Z 460.821,A -85,B 0,C 180,E1 -25531.004,E2 -25531.004} C_VEL
LIN {X 0,Y 132.822,Z 458.076,A -85,B 0,C 180,E1 -25533.274,E2 -25533.274} C_VEL
LIN {X 0,Y 131.226,Z 455.762,A -85,B 0,C 180,E1 -25535.566,E2 -25535.566} C_VEL
LIN {X 0,Y 130.677,Z 454.293,A -85,B 0,C 180,E1 -25536.677,E2 -25536.677} C_VEL
LIN {X 0,Y 127.522,Z 450.633,A -85,B 0,C 180,E1 -25541.735,E2 -25541.735} C_VEL
LIN {X 0,Y 126.857,Z 448.592,A -85,B 0,C 180,E1 -25543.507,E2 -25543.507} C_VEL
LIN {X 0,Y 123.057,Z 443.72,A -85,B 0,C 180,E1 -25558.775,E2 -25558.775} C_VEL
LIN {X 0,Y 123.112,Z 443.339,A -85,B 0,C 180,E1 -25560.206,E2 -25560.206} C_VEL
LIN {X 0,Y 127.11,Z 449.288,A -85,B 0,C 180,E1 -25576.36,E2 -25576.36} C_VEL
LIN {X 0,Y 128.099,Z 452.236,A -85,B 0,C 180,E1 -25578.805,E2 -25578.805} C_VEL
LIN {X 0,Y 130.261,Z 455.033,A -85,B 0,C 180,E1 -25582.191,E2 -25582.191} C_VEL
LIN {X 0,Y 133.11,Z 460.458,A -85,B 0,C 180,E1 -25586.668,E2 -25586.668} C_VEL
LIN {X 0,Y 133.693,Z 461.216,A -85,B 0,C 180,E1 -25587.387,E2 -25587.387} C_VEL
LIN {X 0,Y 136.329,Z 466.864,A -85,B 0,C 180,E1 -25591.034,E2 -25591.034} C_VEL
LIN {X 0,Y 139.438,Z 475.064,A -85,B 0,C 180,E1 -25595.603,E2 -25595.603} C_VEL
LIN {X 0,Y 141.022,Z 481.153,A -85,B 0,C 180,E1 -25598.534,E2 -25598.534} C_VEL
LIN {X 0,Y 141.868,Z 487.59,A -85,B 0,C 180,E1 -25601.215,E2 -25601.215} C_VEL
LIN {X 0,Y 141.946,Z 495.76,A -85,B 0,C 180,E1 -25604.432,E2 -25604.432} C_VEL
LIN {X 0,Y 141.02,Z 505.404,A -85,B 0,C 180,E1 -25608.381,E2 -25608.381} C_VEL
LIN {X 0,Y 139.495,Z 513.307,A -85,B 0,C 180,E1 -25611.891,E2 -25611.891} C_VEL
LIN {X 0,Y 138.198,Z 516.578,A -85,B 0,C 180,E1 -25613.307,E2 -25613.307} C_VEL
LIN {X 0,Y 133.237,Z 524.905,A -85,B 0,C 180,E1 -25617.272,E2 -25617.272} C_VEL
LIN {X 0,Y 129.777,Z 530.568,A -85,B 0,C 180,E1 -25620.832,E2 -25620.832} C_VEL
LIN {X 0,Y 126.012,Z 536.058,A -85,B 0,C 180,E1 -25625.274,E2 -25625.274} C_VEL
LIN {X 0,Y 123.022,Z 540.384,A -85,B 0,C 180,E1 -25629.955,E2 -25629.955} C_VEL
LIN {X 0,Y 121.621,Z 542.757,A -85,B 0,C 180,E1 -25633.206,E2 -25633.206} C_VEL
LIN {X 0,Y 120.539,Z 544.563,A -85,B 0,C 180,E1 -25636.514,E2 -25636.514} C_VEL
LIN {X 0,Y 119.411,Z 547.025,A -85,B 0,C 180,E1 -25643.24,E2 -25643.24} C_VEL
LIN {X 0,Y 119.231,Z 547.62,A -85,B 0,C 180,E1 -25646.621,E2 -25646.621} C_VEL
LIN {X 0,Y 119.337,Z 547.781,A -85,B 0,C 180,E1 -25650,E2 -25650} C_VEL
LIN {X 0,Y 119.222,Z 547.62,A -85,B 0,C 180,E1 -25653.379,E2 -25653.379} C_VEL
LIN {X 0,Y 119.338,Z 547.022,A -85,B 0,C 180,E1 -25656.764,E2 -25656.764} C_VEL
LIN {X 0,Y 120.539,Z 544.563,A -85,B 0,C 180,E1 -25663.486,E2 -25663.486} C_VEL
LIN {X 0,Y 122.259,Z 541.603,A -85,B 0,C 180,E1 -25668.431,E2 -25668.431} C_VEL
LIN {X 0,Y 124.943,Z 537.612,A -85,B 0,C 180,E1 -25673.187,E2 -25673.187} C_VEL
LIN {X 0,Y 128.405,Z 532.482,A -85,B 0,C 180,E1 -25677.724,E2 -25677.724} C_VEL
LIN {X 0,Y 131.318,Z 527.969,A -85,B 0,C 180,E1 -25680.87,E2 -25680.87} C_VEL
LIN {X 0,Y 134.746,Z 522.274,A -85,B 0,C 180,E1 -25684.103,E2 -25684.103} C_VEL
LIN {X 0,Y 138.148,Z 516.576,A -85,B 0,C 180,E1 -25686.708,E2 -25686.708} C_VEL
LIN {X 0,Y 139.463,Z 513.306,A -85,B 0,C 180,E1 -25688.119,E2 -25688.119} C_VEL
LIN {X 0,Y 141.017,Z 505.408,A -85,B 0,C 180,E1 -25691.618,E2 -25691.618} C_VEL
LIN {X 0,Y 141.829,Z 497.363,A -85,B 0,C 180,E1 -25694.915,E2 -25694.915} C_VEL
LIN {X 0,Y 141.913,Z 490.576,A -85,B 0,C 180,E1 -25697.61,E2 -25697.61} C_VEL
LIN {X 0,Y 141.663,Z 485.051,A -85,B 0,C 180,E1 -25699.837,E2 -25699.837} C_VEL
LIN {X 0,Y 140.258,Z 477.8,A -85,B 0,C 180,E1 -25703.036,E2 -25703.036} C_VEL
LIN {X 0,Y 137.812,Z 470.6,A -85,B 0,C 180,E1 -25706.753,E2 -25706.753} C_VEL
LIN {X 0,Y 135.765,Z 465.746,A -85,B 0,C 180,E1 -25709.705,E2 -25709.705} C_VEL
LIN {X 0,Y 133.695,Z 461.209,A -85,B 0,C 180,E1 -25712.613,E2 -25712.613} C_VEL
LIN {X 0,Y 131.571,Z 457.924,A -85,B 0,C 180,E1 -25715.543,E2 -25715.543} C_VEL
LIN {X 0,Y 130.127,Z 454.888,A -85,B 0,C 180,E1 -25717.993,E2 -25717.993} C_VEL
LIN {X 0,Y 127.586,Z 451.146,A -85,B 0,C 180,E1 -25722.259,E2 -25722.259} C_VEL
LIN {X 0,Y 126.988,Z 449.013,A -85,B 0,C 180,E1 -25723.934,E2 -25723.934} C_VEL
LIN {X 0,Y 123.081,Z 443.541,A -85,B 0,C 180,E1 -25739.385,E2 -25739.385} C_VEL
LIN {X 0,Y 123.121,Z 443.219,A -85,B 0,C 180,E1 -25739.998,E2 -25739.998} C_VEL
LIN {X 0,Y 125.216,Z 447.687,A -85,B 0,C 180,E1 -25753.181,E2 -25753.181} C_VEL
LIN {X 0,Y 125.747,Z 449.133,A -85,B 0,C 180,E1 -25754.84,E2 -25754.84} C_VEL
LIN {X 0,Y 126.053,Z 453.382,A -85,B 0,C 180,E1 -25757.206,E2 -25757.206} C_VEL
LIN {X 0,Y 126.165,Z 457.869,A -85,B 0,C 180,E1 -25759.555,E2 -25759.555} C_VEL
LIN {X 0,Y 126.77,Z 459.669,A -85,B 0,C 180,E1 -25761.164,E2 -25761.164} C_VEL
LIN {X 0,Y 127.688,Z 460.707,A -85,B 0,C 180,E1 -25762.659,E2 -25762.659} C_VEL
LIN {X 0,Y 129.404,Z 463.97,A -85,B 0,C 180,E1 -25765.75,E2 -25765.75} C_VEL
LIN {X 0,Y 130.359,Z 465.443,A -85,B 0,C 180,E1 -25767.273,E2 -25767.273} C_VEL
LIN {X 0,Y 132.783,Z 470.073,A -85,B 0,C 180,E1 -25771.066,E2 -25771.066} C_VEL
LIN {X 0,Y 135.247,Z 475.337,A -85,B 0,C 180,E1 -25774.86,E2 -25774.86} C_VEL
LIN {X 0,Y 138.102,Z 482.805,A -85,B 0,C 180,E1 -25779.503,E2 -25779.503} C_VEL
LIN {X 0,Y 140.311,Z 490.61,A -85,B 0,C 180,E1 -25783.887,E2 -25783.887} C_VEL
LIN {X 0,Y 141.755,Z 498.342,A -85,B 0,C 180,E1 -25788.043,E2 -25788.043} C_VEL
LIN {X 0,Y 142.39,Z 505.972,A -85,B 0,C 180,E1 -25792.156,E2 -25792.156} C_VEL
LIN {X 0,Y 142.898,Z 513.64,A -85,B 0,C 180,E1 -25796.726,E2 -25796.726} C_VEL
LIN {X 0,Y 144.268,Z 519.448,A -85,B 0,C 180,E1 -25800.847,E2 -25800.847} C_VEL
LIN {X 0,Y 146.904,Z 524.803,A -85,B 0,C 180,E1 -25805.36,E2 -25805.36} C_VEL
LIN {X 0,Y 150.285,Z 528.768,A -85,B 0,C 180,E1 -25809.271,E2 -25809.271} C_VEL
LIN {X 0,Y 156.328,Z 533.004,A -85,B 0,C 180,E1 -25814.352,E2 -25814.352} C_VEL
LIN {X 0,Y 161.02,Z 535.165,A -85,B 0,C 180,E1 -25817.395,E2 -25817.395} C_VEL
LIN {X 0,Y 170.233,Z 537.69,A -85,B 0,C 180,E1 -25822.224,E2 -25822.224} C_VEL
LIN {X 0,Y 177.837,Z 538.83,A -85,B 0,C 180,E1 -25825.467,E2 -25825.467} C_VEL
LIN {X 0,Y 184.005,Z 539.228,A -85,B 0,C 180,E1 -25827.811,E2 -25827.811} C_VEL
LIN {X 0,Y 190.105,Z 539.218,A -85,B 0,C 180,E1 -25830,E2 -25830} C_VEL
LIN {X 0,Y 182.909,Z 539.165,A -85,B 0,C 180,E1 -25832.579,E2 -25832.579} C_VEL
LIN {X 0,Y 176.396,Z 538.686,A -85,B 0,C 180,E1 -25835.108,E2 -25835.108} C_VEL
LIN {X 0,Y 166.205,Z 536.776,A -85,B 0,C 180,E1 -25839.738,E2 -25839.738} C_VEL
LIN {X 0,Y 159.16,Z 534.402,A -85,B 0,C 180,E1 -25843.73,E2 -25843.73} C_VEL
LIN {X 0,Y 154.407,Z 531.959,A -85,B 0,C 180,E1 -25847.097,E2 -25847.097} C_VEL
LIN {X 0,Y 148.961,Z 527.404,A -85,B 0,C 180,E1 -25852.175,E2 -25852.175} C_VEL
LIN {X 0,Y 145.15,Z 521.687,A -85,B 0,C 180,E1 -25857.371,E2 -25857.371} C_VEL
LIN {X 0,Y 143.355,Z 515.797,A -85,B 0,C 180,E1 -25861.804,E2 -25861.804} C_VEL
LIN {X 0,Y 142.633,Z 510.277,A -85,B 0,C 180,E1 -25865.376,E2 -25865.376} C_VEL
LIN {X 0,Y 142.302,Z 503.456,A -85,B 0,C 180,E1 -25869.208,E2 -25869.208} C_VEL
LIN {X 0,Y 141.394,Z 496.217,A -85,B 0,C 180,E1 -25873.117,E2 -25873.117} C_VEL
LIN {X 0,Y 140.081,Z 489.576,A -85,B 0,C 180,E1 -25876.698,E2 -25876.698} C_VEL
LIN {X 0,Y 137.639,Z 481.574,A -85,B 0,C 180,E1 -25881.283,E2 -25881.283} C_VEL
LIN {X 0,Y 134.636,Z 474.089,A -85,B 0,C 180,E1 -25886.048,E2 -25886.048} C_VEL
LIN {X 0,Y 132.329,Z 468.944,A -85,B 0,C 180,E1 -25889.701,E2 -25889.701} C_VEL
LIN {X 0,Y 129.416,Z 463.939,A -85,B 0,C 180,E1 -25894.252,E2 -25894.252} C_VEL
LIN {X 0,Y 127.689,Z 460.704,A -85,B 0,C 180,E1 -25897.341,E2 -25897.341} C_VEL
LIN {X 0,Y 125.161,Z 457.448,A -85,B 0,C 180,E1 -25902.015,E2 -25902.015} C_VEL
LIN {X 0,Y 124.641,Z 455.962,A -85,B 0,C 180,E1 -25903.627,E2 -25903.627} C_VEL
LIN {X 0,Y 122.043,Z 453.042,A -85,B 0,C 180,E1 -25911.308,E2 -25911.308} C_VEL
LIN {X 0,Y 121.438,Z 450.401,A -85,B 0,C 180,E1 -25920.209,E2 -25920.209} C_VEL
LIN {X 0,Y 124.454,Z 455.448,A -85,B 0,C 180,E1 -25934.723,E2 -25934.723} C_VEL
LIN {X 0,Y 126.248,Z 459.835,A -85,B 0,C 180,E1 -25939.514,E2 -25939.514} C_VEL
LIN {X 0,Y 127.951,Z 462.615,A -85,B 0,C 180,E1 -25942.614,E2 -25942.614} C_VEL
LIN {X 0,Y 130.198,Z 467.095,A -85,B 0,C 180,E1 -25946.446,E2 -25946.446} C_VEL
LIN {X 0,Y 133.266,Z 475.097,A -85,B 0,C 180,E1 -25951.829,E2 -25951.829} C_VEL
LIN {X 0,Y 134.894,Z 480.436,A -85,B 0,C 180,E1 -25954.969,E2 -25954.969} C_VEL
LIN {X 0,Y 136.062,Z 486.243,A -85,B 0,C 180,E1 -25957.865,E2 -25957.865} C_VEL
LIN {X 0,Y 136.362,Z 492.329,A -85,B 0,C 180,E1 -25960.594,E2 -25960.594} C_VEL
LIN {X 0,Y 135.965,Z 499.433,A -85,B 0,C 180,E1 -25963.644,E2 -25963.644} C_VEL
LIN {X 0,Y 134.99,Z 506.566,A -85,B 0,C 180,E1 -25966.795,E2 -25966.795} C_VEL
LIN {X 0,Y 133.591,Z 513.096,A -85,B 0,C 180,E1 -25969.877,E2 -25969.877} C_VEL
LIN {X 0,Y 132.519,Z 516.379,A -85,B 0,C 180,E1 -25971.455,E2 -25971.455} C_VEL
LIN {X 0,Y 127.292,Z 524.707,A -85,B 0,C 180,E1 -25975.535,E2 -25975.535} C_VEL
LIN {X 0,Y 123.592,Z 530.369,A -85,B 0,C 180,E1 -25979.218,E2 -25979.218} C_VEL
LIN {X 0,Y 119.562,Z 535.859,A -85,B 0,C 180,E1 -25983.842,E2 -25983.842} C_VEL
LIN {X 0,Y 116.357,Z 540.186,A -85,B 0,C 180,E1 -25988.753,E2 -25988.753} C_VEL
LIN {X 0,Y 114.789,Z 542.558,A -85,B 0,C 180,E1 -25992.174,E2 -25992.174} C_VEL
LIN {X 0,Y 113.629,Z 544.365,A -85,B 0,C 180,E1 -25995.677,E2 -25995.677} C_VEL
LIN {X 0,Y 112.334,Z 546.827,A -85,B 0,C 180,E1 -26002.812,E2 -26002.812} C_VEL
LIN {X 0,Y 112.14,Z 547.423,A -85,B 0,C 180,E1 -26006.407,E2 -26006.407} C_VEL
LIN {X 0,Y 112.253,Z 547.584,A -85,B 0,C 180,E1 -26010,E2 -26010} C_VEL
LIN {X 0,Y 112.13,Z 547.422,A -85,B 0,C 180,E1 -26013.593,E2 -26013.593} C_VEL
LIN {X 0,Y 112.275,Z 546.825,A -85,B 0,C 180,E1 -26017.192,E2 -26017.192} C_VEL
LIN {X 0,Y 113.629,Z 544.365,A -85,B 0,C 180,E1 -26024.323,E2 -26024.323} C_VEL
LIN {X 0,Y 115.509,Z 541.405,A -85,B 0,C 180,E1 -26029.55,E2 -26029.55} C_VEL
LIN {X 0,Y 118.431,Z 537.414,A -85,B 0,C 180,E1 -26034.544,E2 -26034.544} C_VEL
LIN {X 0,Y 122.156,Z 532.284,A -85,B 0,C 180,E1 -26039.276,E2 -26039.276} C_VEL
LIN {X 0,Y 124.893,Z 528.318,A -85,B 0,C 180,E1 -26042.198,E2 -26042.198} C_VEL
LIN {X 0,Y 128.914,Z 522.076,A -85,B 0,C 180,E1 -26045.877,E2 -26045.877} C_VEL
LIN {X 0,Y 132.449,Z 516.376,A -85,B 0,C 180,E1 -26048.57,E2 -26048.57} C_VEL
LIN {X 0,Y 133.59,Z 513.096,A -85,B 0,C 180,E1 -26050.124,E2 -26050.124} C_VEL
LIN {X 0,Y 135.127,Z 505.79,A -85,B 0,C 180,E1 -26053.558,E2 -26053.558} C_VEL
LIN {X 0,Y 135.965,Z 499.433,A -85,B 0,C 180,E1 -26056.356,E2 -26056.356} C_VEL
LIN {X 0,Y 136.322,Z 492.41,A -85,B 0,C 180,E1 -26059.392,E2 -26059.392} C_VEL
LIN {X 0,Y 136.052,Z 486.245,A -85,B 0,C 180,E1 -26062.14,E2 -26062.14} C_VEL
LIN {X 0,Y 134.888,Z 480.451,A -85,B 0,C 180,E1 -26065.029,E2 -26065.029} C_VEL
LIN {X 0,Y 133.266,Z 475.098,A -85,B 0,C 180,E1 -26068.17,E2 -26068.17} C_VEL
LIN {X 0,Y 131.403,Z 470.439,A -85,B 0,C 180,E1 -26071.224,E2 -26071.224} C_VEL
LIN {X 0,Y 130.211,Z 467.063,A -85,B 0,C 180,E1 -26073.556,E2 -26073.556} C_VEL
LIN {X 0,Y 127.124,Z 461.002,A -85,B 0,C 180,E1 -26078.938,E2 -26078.938} C_VEL
LIN {X 0,Y 125.405,Z 458.326,A -85,B 0,C 180,E1 -26082.308,E2 -26082.308} C_VEL
LIN {X 0,Y 124.458,Z 455.436,A -85,B 0,C 180,E1 -26085.277,E2 -26085.277} C_VEL
LIN {X 0,Y 121.453,Z 450.326,A -85,B 0,C 180,E1 -26099.998,E2 -26099.998} C_VEL
LIN {X 0,Y 123.367,Z 454.584,A -85,B 0,C 180,E1 -26113.17,E2 -26113.17} C_VEL
LIN {X 0,Y 124.707,Z 456.277,A -85,B 0,C 180,E1 -26116.658,E2 -26116.658} C_VEL
LIN {X 0,Y 125.886,Z 458.611,A -85,B 0,C 180,E1 -26119.569,E2 -26119.569} C_VEL
LIN {X 0,Y 126.77,Z 459.669,A -85,B 0,C 180,E1 -26121.164,E2 -26121.164} C_VEL
LIN {X 0,Y 127.618,Z 461.167,A -85,B 0,C 180,E1 -26122.753,E2 -26122.753} C_VEL
LIN {X 0,Y 128.38,Z 464.407,A -85,B 0,C 180,E1 -26124.94,E2 -26124.94} C_VEL
LIN {X 0,Y 129.213,Z 476.217,A -85,B 0,C 180,E1 -26131.062,E2 -26131.062} C_VEL
LIN {X 0,Y 129.846,Z 478.365,A -85,B 0,C 180,E1 -26132.546,E2 -26132.546} C_VEL
LIN {X 0,Y 131.622,Z 483.141,A -85,B 0,C 180,E1 -26135.967,E2 -26135.967} C_VEL
LIN {X 0,Y 133.848,Z 490.752,A -85,B 0,C 180,E1 -26140.866,E2 -26140.866} C_VEL
LIN {X 0,Y 135.335,Z 498.606,A -85,B 0,C 180,E1 -26145.561,E2 -26145.561} C_VEL
LIN {X 0,Y 136.001,Z 505.743,A -85,B 0,C 180,E1 -26149.755,E2 -26149.755} C_VEL
LIN {X 0,Y 136.074,Z 513.364,A -85,B 0,C 180,E1 -26154.477,E2 -26154.477} C_VEL
LIN {X 0,Y 136.94,Z 519.683,A -85,B 0,C 180,E1 -26159.123,E2 -26159.123} C_VEL
LIN {X 0,Y 139.216,Z 525.302,A -85,B 0,C 180,E1 -26164.128,E2 -26164.128} C_VEL
LIN {X 0,Y 141.906,Z 529.038,A -85,B 0,C 180,E1 -26168.006,E2 -26168.006} C_VEL
LIN {X 0,Y 146.967,Z 533.012,A -85,B 0,C 180,E1 -26173.014,E2 -26173.014} C_VEL
LIN {X 0,Y 151.795,Z 535.428,A -85,B 0,C 180,E1 -26176.615,E2 -26176.615} C_VEL
LIN {X 0,Y 157.071,Z 537.133,A -85,B 0,C 180,E1 -26179.847,E2 -26179.847} C_VEL
LIN {X 0,Y 169.159,Z 539.162,A -85,B 0,C 180,E1 -26185.63,E2 -26185.63} C_VEL
LIN {X 0,Y 175.779,Z 539.561,A -85,B 0,C 180,E1 -26188.232,E2 -26188.232} C_VEL
LIN {X 0,Y 180.627,Z 539.477,A -85,B 0,C 180,E1 -26190,E2 -26190} C_VEL
LIN {X 0,Y 174.316,Z 539.496,A -85,B 0,C 180,E1 -26192.311,E2 -26192.311} C_VEL
LIN {X 0,Y 168.165,Z 539.095,A -85,B 0,C 180,E1 -26194.795,E2 -26194.795} C_VEL
LIN {X 0,Y 156.747,Z 537.037,A -85,B 0,C 180,E1 -26200.331,E2 -26200.331} C_VEL
LIN {X 0,Y 149.495,Z 534.38,A -85,B 0,C 180,E1 -26204.983,E2 -26204.983} C_VEL
LIN {X 0,Y 143.738,Z 530.677,A -85,B 0,C 180,E1 -26210.014,E2 -26210.014} C_VEL
LIN {X 0,Y 139.677,Z 526.095,A -85,B 0,C 180,E1 -26215.087,E2 -26215.087} C_VEL
LIN {X 0,Y 137.417,Z 521.188,A -85,B 0,C 180,E1 -26219.61,E2 -26219.61} C_VEL
LIN {X 0,Y 136.205,Z 515.031,A -85,B 0,C 180,E1 -26224.356,E2 -26224.356} C_VEL
LIN {X 0,Y 136.042,Z 508.919,A -85,B 0,C 180,E1 -26228.31,E2 -26228.31} C_VEL
LIN {X 0,Y 135.92,Z 504.045,A -85,B 0,C 180,E1 -26231.25,E2 -26231.25} C_VEL
LIN {X 0,Y 135.115,Z 497,A -85,B 0,C 180,E1 -26235.401,E2 -26235.401} C_VEL
LIN {X 0,Y 133.499,Z 489.544,A -85,B 0,C 180,E1 -26239.937,E2 -26239.937} C_VEL
LIN {X 0,Y 131.135,Z 481.807,A -85,B 0,C 180,E1 -26245.012,E2 -26245.012} C_VEL
LIN {X 0,Y 128.28,Z 474.566,A -85,B 0,C 180,E1 -26250.459,E2 -26250.459} C_VEL
LIN {X 0,Y 126.602,Z 471.109,A -85,B 0,C 180,E1 -26253.636,E2 -26253.636} C_VEL
LIN {X 0,Y 124.236,Z 466.595,A -85,B 0,C 180,E1 -26258.428,E2 -26258.428} C_VEL
LIN {X 0,Y 122.22,Z 463.315,A -85,B 0,C 180,E1 -26263.293,E2 -26263.293} C_VEL
LIN {X 0,Y 121.098,Z 461.414,A -85,B 0,C 180,E1 -26266.579,E2 -26266.579} C_VEL
LIN {X 0,Y 119.463,Z 457.299,A -85,B 0,C 180,E1 -26280.002,E2 -26280.002} C_VEL
LIN {X 0,Y 121.519,Z 461.713,A -85,B 0,C 180,E1 -26293.378,E2 -26293.378} C_VEL
LIN {X 0,Y 122.05,Z 462.811,A -85,B 0,C 180,E1 -26295.02,E2 -26295.02} C_VEL
LIN {X 0,Y 123.044,Z 465.526,A -85,B 0,C 180,E1 -26298.043,E2 -26298.043} C_VEL
LIN {X 0,Y 124.543,Z 468.383,A -85,B 0,C 180,E1 -26301.52,E2 -26301.52} C_VEL
LIN {X 0,Y 126.387,Z 472.779,A -85,B 0,C 180,E1 -26305.53,E2 -26305.53} C_VEL
LIN {X 0,Y 128.551,Z 479.431,A -85,B 0,C 180,E1 -26310.38,E2 -26310.38} C_VEL
LIN {X 0,Y 130.093,Z 485.087,A -85,B 0,C 180,E1 -26313.929,E2 -26313.929} C_VEL
LIN {X 0,Y 130.786,Z 491.089,A -85,B 0,C 180,E1 -26317.197,E2 -26317.197} C_VEL
LIN {X 0,Y 130.688,Z 496.366,A -85,B 0,C 180,E1 -26319.702,E2 -26319.702} C_VEL
LIN {X 0,Y 129.87,Z 503.617,A -85,B 0,C 180,E1 -26323.068,E2 -26323.068} C_VEL
LIN {X 0,Y 128.26,Z 511.421,A -85,B 0,C 180,E1 -26326.892,E2 -26326.892} C_VEL
LIN {X 0,Y 126.858,Z 516.175,A -85,B 0,C 180,E1 -26329.388,E2 -26329.388} C_VEL
LIN {X 0,Y 124.168,Z 520.504,A -85,B 0,C 180,E1 -26331.494,E2 -26331.494} C_VEL
LIN {X 0,Y 120.635,Z 525.665,A -85,B 0,C 180,E1 -26334.369,E2 -26334.369} C_VEL
LIN {X 0,Y 116.001,Z 532.087,A -85,B 0,C 180,E1 -26339.005,E2 -26339.005} C_VEL
LIN {X 0,Y 111.986,Z 537.217,A -85,B 0,C 180,E1 -26343.941,E2 -26343.941} C_VEL
LIN {X 0,Y 108.819,Z 541.207,A -85,B 0,C 180,E1 -26349.194,E2 -26349.194} C_VEL
LIN {X 0,Y 106.718,Z 544.167,A -85,B 0,C 180,E1 -26354.727,E2 -26354.727} C_VEL
LIN {X 0,Y 105.277,Z 546.629,A -85,B 0,C 180,E1 -26362.327,E2 -26362.327} C_VEL
LIN {X 0,Y 105.048,Z 547.226,A -85,B 0,C 180,E1 -26366.164,E2 -26366.164} C_VEL
LIN {X 0,Y 105.171,Z 547.388,A -85,B 0,C 180,E1 -26370,E2 -26370} C_VEL
LIN {X 0,Y 105.039,Z 547.225,A -85,B 0,C 180,E1 -26373.836,E2 -26373.836} C_VEL
LIN {X 0,Y 105.233,Z 546.628,A -85,B 0,C 180,E1 -26377.676,E2 -26377.676} C_VEL
LIN {X 0,Y 106.718,Z 544.167,A -85,B 0,C 180,E1 -26385.273,E2 -26385.273} C_VEL
LIN {X 0,Y 108.819,Z 541.207,A -85,B 0,C 180,E1 -26390.806,E2 -26390.806} C_VEL
LIN {X 0,Y 111.997,Z 537.217,A -85,B 0,C 180,E1 -26396.056,E2 -26396.056} C_VEL
LIN {X 0,Y 116.004,Z 532.087,A -85,B 0,C 180,E1 -26400.994,E2 -26400.994} C_VEL
LIN {X 0,Y 119.877,Z 526.676,A -85,B 0,C 180,E1 -26404.989,E2 -26404.989} C_VEL
LIN {X 0,Y 124.125,Z 520.503,A -85,B 0,C 180,E1 -26408.521,E2 -26408.521} C_VEL
LIN {X 0,Y 126.818,Z 516.173,A -85,B 0,C 180,E1 -26410.628,E2 -26410.628} C_VEL
LIN {X 0,Y 128.759,Z 509.346,A -85,B 0,C 180,E1 -26414.164,E2 -26414.164} C_VEL
LIN {X 0,Y 130.342,Z 500.233,A -85,B 0,C 180,E1 -26418.492,E2 -26418.492} C_VEL
LIN {X 0,Y 130.852,Z 493.092,A -85,B 0,C 180,E1 -26421.853,E2 -26421.853} C_VEL
LIN {X 0,Y 130.503,Z 487.627,A -85,B 0,C 180,E1 -26424.596,E2 -26424.596} C_VEL
LIN {X 0,Y 129.282,Z 481.887,A -85,B 0,C 180,E1 -26427.991,E2 -26427.991} C_VEL
LIN {X 0,Y 127.658,Z 476.436,A -85,B 0,C 180,E1 -26431.743,E2 -26431.743} C_VEL
LIN {X 0,Y 125.966,Z 471.91,A -85,B 0,C 180,E1 -26435.262,E2 -26435.262} C_VEL
LIN {X 0,Y 123.87,Z 466.892,A -85,B 0,C 180,E1 -26440.096,E2 -26440.096} C_VEL
LIN {X 0,Y 122.519,Z 464.401,A -85,B 0,C 180,E1 -26443.331,E2 -26443.331} C_VEL
LIN {X 0,Y 122.052,Z 462.803,A -85,B 0,C 180,E1 -26444.98,E2 -26444.98} C_VEL
LIN {X 0,Y 121.518,Z 461.717,A -85,B 0,C 180,E1 -26446.622,E2 -26446.622} C_VEL
LIN {X 0,Y 119.473,Z 457.269,A -85,B 0,C 180,E1 -26459.998,E2 -26459.998} C_VEL
LIN {X 0,Y 121.096,Z 461.421,A -85,B 0,C 180,E1 -26473.422,E2 -26473.422} C_VEL
LIN {X 0,Y 122.766,Z 464.527,A -85,B 0,C 180,E1 -26478.35,E2 -26478.35} C_VEL
LIN {X 0,Y 124.242,Z 466.582,A -85,B 0,C 180,E1 -26481.571,E2 -26481.571} C_VEL
LIN {X 0,Y 126.601,Z 471.112,A -85,B 0,C 180,E1 -26486.364,E2 -26486.364} C_VEL
LIN {X 0,Y 128.648,Z 475.606,A -85,B 0,C 180,E1 -26490.351,E2 -26490.351} C_VEL
LIN {X 0,Y 129.846,Z 478.365,A -85,B 0,C 180,E1 -26492.546,E2 -26492.546} C_VEL
LIN {X 0,Y 130.541,Z 480.491,A -85,B 0,C 180,E1 -26493.971,E2 -26493.971} C_VEL
LIN {X 0,Y 130.705,Z 482.996,A -85,B 0,C 180,E1 -26495.306,E2 -26495.306} C_VEL
LIN {X 0,Y 130.254,Z 488.581,A -85,B 0,C 180,E1 -26497.786,E2 -26497.786} C_VEL
LIN {X 0,Y 129.007,Z 497,A -85,B 0,C 180,E1 -26501.642,E2 -26501.642} C_VEL
LIN {X 0,Y 129.052,Z 499.39,A -85,B 0,C 180,E1 -26503.086,E2 -26503.086} C_VEL
LIN {X 0,Y 129.631,Z 506.079,A -85,B 0,C 180,E1 -26507.394,E2 -26507.394} C_VEL
LIN {X 0,Y 129.629,Z 512.248,A -85,B 0,C 180,E1 -26511.43,E2 -26511.43} C_VEL
LIN {X 0,Y 129.849,Z 519.914,A -85,B 0,C 180,E1 -26517.232,E2 -26517.232} C_VEL
LIN {X 0,Y 130.93,Z 524.241,A -85,B 0,C 180,E1 -26521.113,E2 -26521.113} C_VEL
LIN {X 0,Y 133.909,Z 529.465,A -85,B 0,C 180,E1 -26526.82,E2 -26526.82} C_VEL
LIN {X 0,Y 138.629,Z 533.512,A -85,B 0,C 180,E1 -26532.292,E2 -26532.292} C_VEL
LIN {X 0,Y 144.285,Z 536.273,A -85,B 0,C 180,E1 -26536.944,E2 -26536.944} C_VEL
LIN {X 0,Y 152.656,Z 538.493,A -85,B 0,C 180,E1 -26542.061,E2 -26542.061} C_VEL
LIN {X 0,Y 161.951,Z 539.59,A -85,B 0,C 180,E1 -26546.446,E2 -26546.446} C_VEL
LIN {X 0,Y 171.02,Z 539.738,A -85,B 0,C 180,E1 -26550,E2 -26550} C_VEL
LIN {X 0,Y 161.95,Z 539.591,A -85,B 0,C 180,E1 -26553.55,E2 -26553.55} C_VEL
LIN {X 0,Y 152.653,Z 538.493,A -85,B 0,C 180,E1 -26557.939,E2 -26557.939} C_VEL
LIN {X 0,Y 144.286,Z 536.272,A -85,B 0,C 180,E1 -26563.056,E2 -26563.056} C_VEL
LIN {X 0,Y 137.062,Z 532.449,A -85,B 0,C 180,E1 -26569.362,E2 -26569.362} C_VEL
LIN {X 0,Y 132.465,Z 527.379,A -85,B 0,C 180,E1 -26575.589,E2 -26575.589} C_VEL
LIN {X 0,Y 130.454,Z 522.531,A -85,B 0,C 180,E1 -26580.465,E2 -26580.465} C_VEL
LIN {X 0,Y 129.575,Z 516.41,A -85,B 0,C 180,E1 -26585.556,E2 -26585.556} C_VEL
LIN {X 0,Y 129.699,Z 510.389,A -85,B 0,C 180,E1 -26589.76,E2 -26589.76} C_VEL
LIN {X 0,Y 129.511,Z 504.245,A -85,B 0,C 180,E1 -26593.81,E2 -26593.81} C_VEL
LIN {X 0,Y 128.917,Z 498.175,A -85,B 0,C 180,E1 -26597.732,E2 -26597.732} C_VEL
LIN {X 0,Y 127.425,Z 490.939,A -85,B 0,C 180,E1 -26602.651,E2 -26602.651} C_VEL
LIN {X 0,Y 125.393,Z 484.03,A -85,B 0,C 180,E1 -26607.829,E2 -26607.829} C_VEL
LIN {X 0,Y 124.061,Z 480.149,A -85,B 0,C 180,E1 -26611.129,E2 -26611.129} C_VEL
LIN {X 0,Y 122.567,Z 476.615,A -85,B 0,C 180,E1 -26614.531,E2 -26614.531} C_VEL
LIN {X 0,Y 120.642,Z 472.401,A -85,B 0,C 180,E1 -26619.543,E2 -26619.543} C_VEL
LIN {X 0,Y 118.403,Z 468.264,A -85,B 0,C 180,E1 -26626.267,E2 -26626.267} C_VEL
LIN {X 0,Y 116.887,Z 465.054,A -85,B 0,C 180,E1 -26636.555,E2 -26636.555} C_VEL
LIN {X 0,Y 117.131,Z 464.104,A -85,B 0,C 180,E1 -26640.002,E2 -26640.002} C_VEL
LIN {X 0,Y 117.929,Z 467.318,A -85,B 0,C 180,E1 -26650.301,E2 -26650.301} C_VEL
LIN {X 0,Y 118.9,Z 468.657,A -85,B 0,C 180,E1 -26653.678,E2 -26653.678} C_VEL
LIN {X 0,Y 120.933,Z 474.051,A -85,B 0,C 180,E1 -26660.409,E2 -26660.409} C_VEL
LIN {X 0,Y 122.081,Z 477.456,A -85,B 0,C 180,E1 -26663.766,E2 -26663.766} C_VEL
LIN {X 0,Y 123.995,Z 484.176,A -85,B 0,C 180,E1 -26669.171,E2 -26669.171} C_VEL
LIN {X 0,Y 125.13,Z 490,A -85,B 0,C 180,E1 -26673.206,E2 -26673.206} C_VEL
LIN {X 0,Y 125.429,Z 494.67,A -85,B 0,C 180,E1 -26675.864,E2 -26675.864} C_VEL
LIN {X 0,Y 124.941,Z 500.36,A -85,B 0,C 180,E1 -26678.826,E2 -26678.826} C_VEL
LIN {X 0,Y 123.634,Z 507.294,A -85,B 0,C 180,E1 -26682.356,E2 -26682.356} C_VEL
LIN {X 0,Y 122.134,Z 513.061,A -85,B 0,C 180,E1 -26685.454,E2 -26685.454} C_VEL
LIN {X 0,Y 120.594,Z 517.544,A -85,B 0,C 180,E1 -26687.919,E2 -26687.919} C_VEL
LIN {X 0,Y 114.922,Z 525.468,A -85,B 0,C 180,E1 -26692.3,E2 -26692.3} C_VEL
LIN {X 0,Y 111.562,Z 529.973,A -85,B 0,C 180,E1 -26695.462,E2 -26695.462} C_VEL
LIN {X 0,Y 106.919,Z 535.463,A -85,B 0,C 180,E1 -26700.463,E2 -26700.463} C_VEL
LIN {X 0,Y 103.226,Z 539.791,A -85,B 0,C 180,E1 -26705.89,E2 -26705.89} C_VEL
LIN {X 0,Y 101.273,Z 542.162,A -85,B 0,C 180,E1 -26709.698,E2 -26709.698} C_VEL
LIN {X 0,Y 99.842,Z 543.968,A -85,B 0,C 180,E1 -26713.647,E2 -26713.647} C_VEL
LIN {X 0,Y 98.224,Z 546.432,A -85,B 0,C 180,E1 -26721.773,E2 -26721.773} C_VEL
LIN {X 0,Y 97.954,Z 547.028,A -85,B 0,C 180,E1 -26725.886,E2 -26725.886} C_VEL
LIN {X 0,Y 98.077,Z 547.191,A -85,B 0,C 180,E1 -26730,E2 -26730} C_VEL
LIN {X 0,Y 97.945,Z 547.028,A -85,B 0,C 180,E1 -26734.115,E2 -26734.115} C_VEL
LIN {X 0,Y 98.191,Z 546.431,A -85,B 0,C 180,E1 -26738.23,E2 -26738.23} C_VEL
LIN {X 0,Y 99.842,Z 543.968,A -85,B 0,C 180,E1 -26746.353,E2 -26746.353} C_VEL
LIN {X 0,Y 102.196,Z 541.01,A -85,B 0,C 180,E1 -26752.224,E2 -26752.224} C_VEL
LIN {X 0,Y 105.65,Z 537.02,A -85,B 0,C 180,E1 -26757.752,E2 -26757.752} C_VEL
LIN {X 0,Y 109.966,Z 531.889,A -85,B 0,C 180,E1 -26762.904,E2 -26762.904} C_VEL
LIN {X 0,Y 114.884,Z 525.466,A -85,B 0,C 180,E1 -26767.715,E2 -26767.715} C_VEL
LIN {X 0,Y 120.56,Z 517.543,A -85,B 0,C 180,E1 -26772.096,E2 -26772.096} C_VEL
LIN {X 0,Y 122.901,Z 510.454,A -85,B 0,C 180,E1 -26776.024,E2 -26776.024} C_VEL
LIN {X 0,Y 124.772,Z 501.741,A -85,B 0,C 180,E1 -26780.504,E2 -26780.504} C_VEL
LIN {X 0,Y 125.443,Z 494.637,A -85,B 0,C 180,E1 -26784.147,E2 -26784.147} C_VEL
LIN {X 0,Y 125.109,Z 490.039,A -85,B 0,C 180,E1 -26786.788,E2 -26786.788} C_VEL
LIN {X 0,Y 123.99,Z 484.186,A -85,B 0,C 180,E1 -26790.828,E2 -26790.828} C_VEL
LIN {X 0,Y 122.075,Z 477.467,A -85,B 0,C 180,E1 -26796.232,E2 -26796.232} C_VEL
LIN {X 0,Y 120.933,Z 474.051,A -85,B 0,C 180,E1 -26799.591,E2 -26799.591} C_VEL
LIN {X 0,Y 118.902,Z 468.653,A -85,B 0,C 180,E1 -26806.322,E2 -26806.322} C_VEL
LIN {X 0,Y 117.239,Z 466.288,A -85,B 0,C 180,E1 -26813.112,E2 -26813.112} C_VEL
LIN {X 0,Y 117.137,Z 464.088,A -85,B 0,C 180,E1 -26819.998,E2 -26819.998} C_VEL
LIN {X 0,Y 117.555,Z 467.015,A -85,B 0,C 180,E1 -26830.33,E2 -26830.33} C_VEL
LIN {X 0,Y 118.406,Z 468.257,A -85,B 0,C 180,E1 -26833.732,E2 -26833.732} C_VEL
LIN {X 0,Y 120.644,Z 472.395,A -85,B 0,C 180,E1 -26840.456,E2 -26840.456} C_VEL
LIN {X 0,Y 122.551,Z 476.647,A -85,B 0,C 180,E1 -26845.472,E2 -26845.472} C_VEL
LIN {X 0,Y 124.071,Z 480.128,A -85,B 0,C 180,E1 -26848.868,E2 -26848.868} C_VEL
LIN {X 0,Y 126.111,Z 486.12,A -85,B 0,C 180,E1 -26853.866,E2 -26853.866} C_VEL
LIN {X 0,Y 127.469,Z 490.868,A -85,B 0,C 180,E1 -26857.334,E2 -26857.334} C_VEL
LIN {X 0,Y 128.914,Z 498.166,A -85,B 0,C 180,E1 -26862.26,E2 -26862.26} C_VEL
LIN {X 0,Y 129.052,Z 499.39,A -85,B 0,C 180,E1 -26863.086,E2 -26863.086} C_VEL
LIN {X 0,Y 129.003,Z 501.811,A -85,B 0,C 180,E1 -26864.499,E2 -26864.499} C_VEL
LIN {X 0,Y 128.426,Z 504.451,A -85,B 0,C 180,E1 -26865.82,E2 -26865.82} C_VEL
LIN {X 0,Y 126.36,Z 509.587,A -85,B 0,C 180,E1 -26868.347,E2 -26868.347} C_VEL
LIN {X 0,Y 123.638,Z 515.845,A -85,B 0,C 180,E1 -26871.74,E2 -26871.74} C_VEL
LIN {X 0,Y 122.972,Z 518.973,A -85,B 0,C 180,E1 -26874.094,E2 -26874.094} C_VEL
LIN {X 0,Y 123.613,Z 524.475,A -85,B 0,C 180,E1 -26879.224,E2 -26879.224} C_VEL
LIN {X 0,Y 126.089,Z 529.924,A -85,B 0,C 180,E1 -26885.549,E2 -26885.549} C_VEL
LIN {X 0,Y 128.163,Z 532.339,A -85,B 0,C 180,E1 -26888.778,E2 -26888.778} C_VEL
LIN {X 0,Y 133.719,Z 535.945,A -85,B 0,C 180,E1 -26894.765,E2 -26894.765} C_VEL
LIN {X 0,Y 142.311,Z 538.584,A -85,B 0,C 180,E1 -26900.992,E2 -26900.992} C_VEL
LIN {X 0,Y 148.803,Z 539.626,A -85,B 0,C 180,E1 -26904.58,E2 -26904.58} C_VEL
LIN {X 0,Y 154.905,Z 540.028,A -85,B 0,C 180,E1 -26907.4,E2 -26907.4} C_VEL
LIN {X 0,Y 161.365,Z 540.001,A -85,B 0,C 180,E1 -26910,E2 -26910} C_VEL
LIN {X 0,Y 154.778,Z 540.021,A -85,B 0,C 180,E1 -26912.653,E2 -26912.653} C_VEL
LIN {X 0,Y 148.308,Z 539.591,A -85,B 0,C 180,E1 -26915.665,E2 -26915.665} C_VEL
LIN {X 0,Y 138.106,Z 537.557,A -85,B 0,C 180,E1 -26921.745,E2 -26921.745} C_VEL
LIN {X 0,Y 132.115,Z 535.061,A -85,B 0,C 180,E1 -26926.765,E2 -26926.765} C_VEL
LIN {X 0,Y 127.142,Z 531.171,A -85,B 0,C 180,E1 -26932.763,E2 -26932.763} C_VEL
LIN {X 0,Y 124.93,Z 528.136,A -85,B 0,C 180,E1 -26936.746,E2 -26936.746} C_VEL
LIN {X 0,Y 123.236,Z 522.371,A -85,B 0,C 180,E1 -26942.802,E2 -26942.802} C_VEL
LIN {X 0,Y 123.065,Z 516.455,A -85,B 0,C 180,E1 -26947.892,E2 -26947.892} C_VEL
LIN {X 0,Y 123.44,Z 510.566,A -85,B 0,C 180,E1 -26952.259,E2 -26952.259} C_VEL
LIN {X 0,Y 123.286,Z 504.199,A -85,B 0,C 180,E1 -26956.84,E2 -26956.84} C_VEL
LIN {X 0,Y 122.696,Z 498.569,A -85,B 0,C 180,E1 -26960.947,E2 -26960.947} C_VEL
LIN {X 0,Y 121.175,Z 491.088,A -85,B 0,C 180,E1 -26966.82,E2 -26966.82} C_VEL
LIN {X 0,Y 119.523,Z 485.344,A -85,B 0,C 180,E1 -26971.942,E2 -26971.942} C_VEL
LIN {X 0,Y 118.434,Z 482.053,A -85,B 0,C 180,E1 -26975.458,E2 -26975.458} C_VEL
LIN {X 0,Y 116.707,Z 477.996,A -85,B 0,C 180,E1 -26980.66,E2 -26980.66} C_VEL
LIN {X 0,Y 115.387,Z 474.97,A -85,B 0,C 180,E1 -26985.901,E2 -26985.901} C_VEL
LIN {X 0,Y 114.164,Z 472.598,A -85,B 0,C 180,E1 -26992.93,E2 -26992.93} C_VEL
LIN {X 0,Y 114.29,Z 470.711,A -85,B 0,C 180,E1 -27000.002,E2 -27000.002} C_VEL
LIN {X 0,Y 115.083,Z 473.937,A -85,B 0,C 180,E1 -27010.559,E2 -27010.559} C_VEL
LIN {X 0,Y 115.812,Z 475.722,A -85,B 0,C 180,E1 -27014.05,E2 -27014.05} C_VEL
LIN {X 0,Y 117.017,Z 479.538,A -85,B 0,C 180,E1 -27019.291,E2 -27019.291} C_VEL
LIN {X 0,Y 118.015,Z 483.052,A -85,B 0,C 180,E1 -27022.964,E2 -27022.964} C_VEL
LIN {X 0,Y 119.245,Z 488.955,A -85,B 0,C 180,E1 -27028.134,E2 -27028.134} C_VEL
LIN {X 0,Y 120.02,Z 493.924,A -85,B 0,C 180,E1 -27031.806,E2 -27031.806} C_VEL
LIN {X 0,Y 119.911,Z 498.731,A -85,B 0,C 180,E1 -27034.863,E2 -27034.863} C_VEL
LIN {X 0,Y 119.061,Z 504.304,A -85,B 0,C 180,E1 -27037.977,E2 -27037.977} C_VEL
LIN {X 0,Y 117.138,Z 511.471,A -85,B 0,C 180,E1 -27041.939,E2 -27041.939} C_VEL
LIN {X 0,Y 115.11,Z 517.335,A -85,B 0,C 180,E1 -27045.403,E2 -27045.403} C_VEL
LIN {X 0,Y 114.378,Z 518.731,A -85,B 0,C 180,E1 -27046.271,E2 -27046.271} C_VEL
LIN {X 0,Y 109.357,Z 525.269,A -85,B 0,C 180,E1 -27050.01,E2 -27050.01} C_VEL
LIN {X 0,Y 105.742,Z 529.774,A -85,B 0,C 180,E1 -27053.262,E2 -27053.262} C_VEL
LIN {X 0,Y 100.773,Z 535.265,A -85,B 0,C 180,E1 -27058.463,E2 -27058.463} C_VEL
LIN {X 0,Y 96.778,Z 539.594,A -85,B 0,C 180,E1 -27064.17,E2 -27064.17} C_VEL
LIN {X 0,Y 94.609,Z 541.964,A -85,B 0,C 180,E1 -27068.197,E2 -27068.197} C_VEL
LIN {X 0,Y 93.016,Z 543.77,A -85,B 0,C 180,E1 -27072.409,E2 -27072.409} C_VEL
LIN {X 0,Y 91.176,Z 546.234,A -85,B 0,C 180,E1 -27081.132,E2 -27081.132} C_VEL
LIN {X 0,Y 90.883,Z 546.831,A -85,B 0,C 180,E1 -27085.565,E2 -27085.565} C_VEL
LIN {X 0,Y 90.976,Z 546.994,A -85,B 0,C 180,E1 -27090,E2 -27090} C_VEL
LIN {X 0,Y 90.875,Z 546.831,A -85,B 0,C 180,E1 -27094.435,E2 -27094.435} C_VEL
LIN {X 0,Y 91.151,Z 546.233,A -85,B 0,C 180,E1 -27098.871,E2 -27098.871} C_VEL
LIN {X 0,Y 93.016,Z 543.77,A -85,B 0,C 180,E1 -27107.591,E2 -27107.591} C_VEL
LIN {X 0,Y 95.624,Z 540.812,A -85,B 0,C 180,E1 -27113.842,E2 -27113.842} C_VEL
LIN {X 0,Y 99.388,Z 536.821,A -85,B 0,C 180,E1 -27119.668,E2 -27119.668} C_VEL
LIN {X 0,Y 104.058,Z 531.692,A -85,B 0,C 180,E1 -27125.035,E2 -27125.035} C_VEL
LIN {X 0,Y 108.459,Z 526.315,A -85,B 0,C 180,E1 -27129.293,E2 -27129.293} C_VEL
LIN {X 0,Y 113.312,Z 520.107,A -85,B 0,C 180,E1 -27133.019,E2 -27133.019} C_VEL
LIN {X 0,Y 115.117,Z 517.335,A -85,B 0,C 180,E1 -27134.593,E2 -27134.593} C_VEL
LIN {X 0,Y 118.007,Z 508.566,A -85,B 0,C 180,E1 -27139.711,E2 -27139.711} C_VEL
LIN {X 0,Y 119.692,Z 500.718,A -85,B 0,C 180,E1 -27144.041,E2 -27144.041} C_VEL
LIN {X 0,Y 120.055,Z 495.105,A -85,B 0,C 180,E1 -27147.384,E2 -27147.384} C_VEL
LIN {X 0,Y 119.248,Z 488.949,A -85,B 0,C 180,E1 -27151.867,E2 -27151.867} C_VEL
LIN {X 0,Y 118,Z 483.002,A -85,B 0,C 180,E1 -27157.084,E2 -27157.084} C_VEL
LIN {X 0,Y 117.013,Z 479.546,A -85,B 0,C 180,E1 -27160.709,E2 -27160.709} C_VEL
LIN {X 0,Y 115.783,Z 475.525,A -85,B 0,C 180,E1 -27166.209,E2 -27166.209} C_VEL
LIN {X 0,Y 115.084,Z 473.935,A -85,B 0,C 180,E1 -27169.442,E2 -27169.442} C_VEL
LIN {X 0,Y 114.301,Z 470.687,A -85,B 0,C 180,E1 -27179.998,E2 -27179.998} C_VEL
LIN {X 0,Y 114.937,Z 474.098,A -85,B 0,C 180,E1 -27191.951,E2 -27191.951} C_VEL
LIN {X 0,Y 115.729,Z 475.96,A -85,B 0,C 180,E1 -27195.857,E2 -27195.857} C_VEL
LIN {X 0,Y 117.225,Z 479.274,A -85,B 0,C 180,E1 -27201.081,E2 -27201.081} C_VEL
LIN {X 0,Y 118.415,Z 482.086,A -85,B 0,C 180,E1 -27204.546,E2 -27204.546} C_VEL
LIN {X 0,Y 119.574,Z 485.427,A -85,B 0,C 180,E1 -27208.163,E2 -27208.163} C_VEL
LIN {X 0,Y 121.23,Z 491.098,A -85,B 0,C 180,E1 -27213.229,E2 -27213.229} C_VEL
LIN {X 0,Y 122.495,Z 497.261,A -85,B 0,C 180,E1 -27218.077,E2 -27218.077} C_VEL
LIN {X 0,Y 123.154,Z 502.85,A -85,B 0,C 180,E1 -27222.215,E2 -27222.215} C_VEL
LIN {X 0,Y 123.415,Z 507.858,A -85,B 0,C 180,E1 -27225.805,E2 -27225.805} C_VEL
LIN {X 0,Y 123.311,Z 513.014,A -85,B 0,C 180,E1 -27229.479,E2 -27229.479} C_VEL
LIN {X 0,Y 122.972,Z 518.973,A -85,B 0,C 180,E1 -27234.094,E2 -27234.094} C_VEL
LIN {X 0,Y 122.472,Z 521.916,A -85,B 0,C 180,E1 -27236.517,E2 -27236.517} C_VEL
LIN {X 0,Y 120.512,Z 526.667,A -85,B 0,C 180,E1 -27240.538,E2 -27240.538} C_VEL
LIN {X 0,Y 119.348,Z 530.702,A -85,B 0,C 180,E1 -27244.763,E2 -27244.763} C_VEL
LIN {X 0,Y 120.078,Z 532.578,A -85,B 0,C 180,E1 -27247.372,E2 -27247.372} C_VEL
LIN {X 0,Y 124.949,Z 536.198,A -85,B 0,C 180,E1 -27253.667,E2 -27253.667} C_VEL
LIN {X 0,Y 129.443,Z 537.967,A -85,B 0,C 180,E1 -27257.758,E2 -27257.758} C_VEL
LIN {X 0,Y 139.245,Z 539.889,A -85,B 0,C 180,E1 -27264.207,E2 -27264.207} C_VEL
LIN {X 0,Y 147.647,Z 540.374,A -85,B 0,C 180,E1 -27268.32,E2 -27268.32} C_VEL
LIN {X 0,Y 151.618,Z 540.267,A -85,B 0,C 180,E1 -27270,E2 -27270} C_VEL
LIN {X 0,Y 141.053,Z 540.017,A -85,B 0,C 180,E1 -27274.814,E2 -27274.814} C_VEL
LIN {X 0,Y 133.818,Z 539.018,A -85,B 0,C 180,E1 -27279.065,E2 -27279.065} C_VEL
LIN {X 0,Y 129.051,Z 537.814,A -85,B 0,C 180,E1 -27282.582,E2 -27282.582} C_VEL
LIN {X 0,Y 123.237,Z 535.138,A -85,B 0,C 180,E1 -27288.278,E2 -27288.278} C_VEL
LIN {X 0,Y 119.097,Z 531.415,A -85,B 0,C 180,E1 -27294.398,E2 -27294.398} C_VEL
LIN {X 0,Y 116.899,Z 526.729,A -85,B 0,C 180,E1 -27300.524,E2 -27300.524} C_VEL
LIN {X 0,Y 116.31,Z 521.486,A -85,B 0,C 180,E1 -27306.095,E2 -27306.095} C_VEL
LIN {X 0,Y 116.881,Z 515.375,A -85,B 0,C 180,E1 -27311.407,E2 -27311.407} C_VEL
LIN {X 0,Y 117.193,Z 510.945,A -85,B 0,C 180,E1 -27314.992,E2 -27314.992} C_VEL
LIN {X 0,Y 117.17,Z 504.55,A -85,B 0,C 180,E1 -27320.064,E2 -27320.064} C_VEL
LIN {X 0,Y 116.529,Z 498.607,A -85,B 0,C 180,E1 -27325.046,E2 -27325.046} C_VEL
LIN {X 0,Y 115.703,Z 494.271,A -85,B 0,C 180,E1 -27328.916,E2 -27328.916} C_VEL
LIN {X 0,Y 114.773,Z 490.091,A -85,B 0,C 180,E1 -27333.21,E2 -27333.21} C_VEL
LIN {X 0,Y 113.968,Z 487.267,A -85,B 0,C 180,E1 -27336.372,E2 -27336.372} C_VEL
LIN {X 0,Y 112.68,Z 483.494,A -85,B 0,C 180,E1 -27341.831,E2 -27341.831} C_VEL
LIN {X 0,Y 111.961,Z 481.525,A -85,B 0,C 180,E1 -27345.46,E2 -27345.46} C_VEL
LIN {X 0,Y 111.315,Z 480.005,A -85,B 0,C 180,E1 -27349.084,E2 -27349.084} C_VEL
LIN {X 0,Y 111.141,Z 477.178,A -85,B 0,C 180,E1 -27360.002,E2 -27360.002} C_VEL
LIN {X 0,Y 111.722,Z 480.41,A -85,B 0,C 180,E1 -27370.88,E2 -27370.88} C_VEL
LIN {X 0,Y 112.286,Z 482.468,A -85,B 0,C 180,E1 -27374.501,E2 -27374.501} C_VEL
LIN {X 0,Y 112.986,Z 484.955,A -85,B 0,C 180,E1 -27378.122,E2 -27378.122} C_VEL
LIN {X 0,Y 113.599,Z 488.168,A -85,B 0,C 180,E1 -27381.878,E2 -27381.878} C_VEL
LIN {X 0,Y 114.401,Z 493.245,A -85,B 0,C 180,E1 -27386.648,E2 -27386.648} C_VEL
LIN {X 0,Y 114.718,Z 498.466,A -85,B 0,C 180,E1 -27390.945,E2 -27390.945} C_VEL
LIN {X 0,Y 114.397,Z 502.429,A -85,B 0,C 180,E1 -27393.569,E2 -27393.569} C_VEL
LIN {X 0,Y 112.927,Z 508.383,A -85,B 0,C 180,E1 -27397.176,E2 -27397.176} C_VEL
LIN {X 0,Y 109.771,Z 517.122,A -85,B 0,C 180,E1 -27402.586,E2 -27402.586} C_VEL
LIN {X 0,Y 108.253,Z 519.911,A -85,B 0,C 180,E1 -27404.428,E2 -27404.428} C_VEL
LIN {X 0,Y 102.987,Z 526.229,A -85,B 0,C 180,E1 -27408.293,E2 -27408.293} C_VEL
LIN {X 0,Y 98.283,Z 531.493,A -85,B 0,C 180,E1 -27412.569,E2 -27412.569} C_VEL
LIN {X 0,Y 93.22,Z 536.622,A -85,B 0,C 180,E1 -27418.148,E2 -27418.148} C_VEL
LIN {X 0,Y 89.148,Z 540.614,A -85,B 0,C 180,E1 -27424.305,E2 -27424.305} C_VEL
LIN {X 0,Y 86.248,Z 543.572,A -85,B 0,C 180,E1 -27430.978,E2 -27430.978} C_VEL
LIN {X 0,Y 84.156,Z 546.036,A -85,B 0,C 180,E1 -27440.385,E2 -27440.385} C_VEL
LIN {X 0,Y 83.798,Z 546.634,A -85,B 0,C 180,E1 -27445.189,E2 -27445.189} C_VEL
LIN {X 0,Y 83.883,Z 546.797,A -85,B 0,C 180,E1 -27450,E2 -27450} C_VEL
LIN {X 0,Y 83.791,Z 546.634,A -85,B 0,C 180,E1 -27454.811,E2 -27454.811} C_VEL
LIN {X 0,Y 84.137,Z 546.036,A -85,B 0,C 180,E1 -27459.617,E2 -27459.617} C_VEL
LIN {X 0,Y 86.248,Z 543.572,A -85,B 0,C 180,E1 -27469.022,E2 -27469.022} C_VEL
LIN {X 0,Y 89.148,Z 540.614,A -85,B 0,C 180,E1 -27475.695,E2 -27475.695} C_VEL
LIN {X 0,Y 93.241,Z 536.623,A -85,B 0,C 180,E1 -27481.844,E2 -27481.844} C_VEL
LIN {X 0,Y 98.287,Z 531.493,A -85,B 0,C 180,E1 -27487.429,E2 -27487.429} C_VEL
LIN {X 0,Y 102.839,Z 526.341,A -85,B 0,C 180,E1 -27491.651,E2 -27491.651} C_VEL
LIN {X 0,Y 108.204,Z 519.909,A -85,B 0,C 180,E1 -27495.598,E2 -27495.598} C_VEL
LIN {X 0,Y 109.78,Z 517.122,A -85,B 0,C 180,E1 -27497.409,E2 -27497.409} C_VEL
LIN {X 0,Y 112.484,Z 509.862,A -85,B 0,C 180,E1 -27501.963,E2 -27501.963} C_VEL
LIN {X 0,Y 114.154,Z 503.547,A -85,B 0,C 180,E1 -27505.715,E2 -27505.715} C_VEL
LIN {X 0,Y 114.661,Z 500.301,A -85,B 0,C 180,E1 -27507.787,E2 -27507.787} C_VEL
LIN {X 0,Y 114.645,Z 496.431,A -85,B 0,C 180,E1 -27510.63,E2 -27510.63} C_VEL
LIN {X 0,Y 114.21,Z 491.963,A -85,B 0,C 180,E1 -27514.483,E2 -27514.483} C_VEL
LIN {X 0,Y 113.587,Z 488.086,A -85,B 0,C 180,E1 -27518.206,E2 -27518.206} C_VEL
LIN {X 0,Y 112.996,Z 484.939,A -85,B 0,C 180,E1 -27521.879,E2 -27521.879} C_VEL
LIN {X 0,Y 112.02,Z 481.215,A -85,B 0,C 180,E1 -27527.415,E2 -27527.415} C_VEL
LIN {X 0,Y 111.139,Z 479.229,A -85,B 0,C 180,E1 -27532.732,E2 -27532.732} C_VEL
LIN {X 0,Y 111.157,Z 477.15,A -85,B 0,C 180,E1 -27539.998,E2 -27539.998} C_VEL
LIN {X 0,Y 111.315,Z 480.005,A -85,B 0,C 180,E1 -27550.916,E2 -27550.916} C_VEL
LIN {X 0,Y 111.955,Z 481.536,A -85,B 0,C 180,E1 -27554.541,E2 -27554.541} C_VEL
LIN {X 0,Y 113.109,Z 484.752,A -85,B 0,C 180,E1 -27560.17,E2 -27560.17} C_VEL
LIN {X 0,Y 113.952,Z 487.293,A -85,B 0,C 180,E1 -27563.632,E2 -27563.632} C_VEL
LIN {X 0,Y 115.104,Z 491.335,A -85,B 0,C 180,E1 -27568.154,E2 -27568.154} C_VEL
LIN {X 0,Y 116.167,Z 496.298,A -85,B 0,C 180,E1 -27572.988,E2 -27572.988} C_VEL
LIN {X 0,Y 116.972,Z 502.113,A -85,B 0,C 180,E1 -27578.011,E2 -27578.011} C_VEL
LIN {X 0,Y 117.251,Z 508.055,A -85,B 0,C 180,E1 -27582.759,E2 -27582.759} C_VEL
LIN {X 0,Y 117.09,Z 513.517,A -85,B 0,C 180,E1 -27587.065,E2 -27587.065} C_VEL
LIN {X 0,Y 116.359,Z 520.371,A -85,B 0,C 180,E1 -27592.844,E2 -27592.844} C_VEL
LIN {X 0,Y 116.555,Z 525.105,A -85,B 0,C 180,E1 -27597.579,E2 -27597.579} C_VEL
LIN {X 0,Y 118.041,Z 529.777,A -85,B 0,C 180,E1 -27603.258,E2 -27603.258} C_VEL
LIN {X 0,Y 120.078,Z 532.578,A -85,B 0,C 180,E1 -27607.372,E2 -27607.372} C_VEL
LIN {X 0,Y 121.143,Z 534.311,A -85,B 0,C 180,E1 -27610.017,E2 -27610.017} C_VEL
LIN {X 0,Y 121.92,Z 536.927,A -85,B 0,C 180,E1 -27614.523,E2 -27614.523} C_VEL
LIN {X 0,Y 123.65,Z 538.912,A -85,B 0,C 180,E1 -27618.957,E2 -27618.957} C_VEL
LIN {X 0,Y 126.106,Z 539.587,A -85,B 0,C 180,E1 -27621.374,E2 -27621.374} C_VEL
LIN {X 0,Y 135.547,Z 540.56,A -85,B 0,C 180,E1 -27627.028,E2 -27627.028} C_VEL
LIN {X 0,Y 141.91,Z 540.531,A -85,B 0,C 180,E1 -27630,E2 -27630} C_VEL
LIN {X 0,Y 133.833,Z 540.445,A -85,B 0,C 180,E1 -27633.872,E2 -27633.872} C_VEL
LIN {X 0,Y 127.619,Z 539.879,A -85,B 0,C 180,E1 -27637.593,E2 -27637.593} C_VEL
LIN {X 0,Y 120.139,Z 538.068,A -85,B 0,C 180,E1 -27643.532,E2 -27643.532} C_VEL
LIN {X 0,Y 114.809,Z 535.413,A -85,B 0,C 180,E1 -27649.629,E2 -27649.629} C_VEL
LIN {X 0,Y 111.248,Z 531.656,A -85,B 0,C 180,E1 -27656.245,E2 -27656.245} C_VEL
LIN {X 0,Y 109.851,Z 527.434,A -85,B 0,C 180,E1 -27662.157,E2 -27662.157} C_VEL
LIN {X 0,Y 109.726,Z 522.827,A -85,B 0,C 180,E1 -27667.479,E2 -27667.479} C_VEL
LIN {X 0,Y 110.614,Z 516.937,A -85,B 0,C 180,E1 -27673.077,E2 -27673.077} C_VEL
LIN {X 0,Y 111.19,Z 510.923,A -85,B 0,C 180,E1 -27678.404,E2 -27678.404} C_VEL
LIN {X 0,Y 111.224,Z 505.723,A -85,B 0,C 180,E1 -27683.112,E2 -27683.112} C_VEL
LIN {X 0,Y 110.777,Z 500.674,A -85,B 0,C 180,E1 -27687.876,E2 -27687.876} C_VEL
LIN {X 0,Y 109.984,Z 495.465,A -85,B 0,C 180,E1 -27693.455,E2 -27693.455} C_VEL
LIN {X 0,Y 109.137,Z 491.547,A -85,B 0,C 180,E1 -27698.631,E2 -27698.631} C_VEL
LIN {X 0,Y 108.379,Z 488.808,A -85,B 0,C 180,E1 -27703.036,E2 -27703.036} C_VEL
LIN {X 0,Y 107.602,Z 486.256,A -85,B 0,C 180,E1 -27708.702,E2 -27708.702} C_VEL
LIN {X 0,Y 107.701,Z 483.472,A -85,B 0,C 180,E1 -27720.002,E2 -27720.002} C_VEL
LIN {X 0,Y 108.059,Z 486.714,A -85,B 0,C 180,E1 -27731.254,E2 -27731.254} C_VEL
LIN {X 0,Y 108.655,Z 490.124,A -85,B 0,C 180,E1 -27736.924,E2 -27736.924} C_VEL
LIN {X 0,Y 109.136,Z 494.014,A -85,B 0,C 180,E1 -27741.642,E2 -27741.642} C_VEL
LIN {X 0,Y 109.449,Z 498.996,A -85,B 0,C 180,E1 -27746.713,E2 -27746.713} C_VEL
LIN {X 0,Y 109.36,Z 502.719,A -85,B 0,C 180,E1 -27749.873,E2 -27749.873} C_VEL
LIN {X 0,Y 108.561,Z 506.609,A -85,B 0,C 180,E1 -27752.694,E2 -27752.694} C_VEL
LIN {X 0,Y 106.596,Z 512.286,A -85,B 0,C 180,E1 -27756.4,E2 -27756.4} C_VEL
LIN {X 0,Y 103.958,Z 518.311,A -85,B 0,C 180,E1 -27760.489,E2 -27760.489} C_VEL
LIN {X 0,Y 102.228,Z 521.089,A -85,B 0,C 180,E1 -27762.351,E2 -27762.351} C_VEL
LIN {X 0,Y 95.031,Z 528.979,A -85,B 0,C 180,E1 -27767.696,E2 -27767.696} C_VEL
LIN {X 0,Y 88.946,Z 534.87,A -85,B 0,C 180,E1 -27773.659,E2 -27773.659} C_VEL
LIN {X 0,Y 84.162,Z 539.198,A -85,B 0,C 180,E1 -27779.932,E2 -27779.932} C_VEL
LIN {X 0,Y 81.525,Z 541.567,A -85,B 0,C 180,E1 -27784.467,E2 -27784.467} C_VEL
LIN {X 0,Y 79.55,Z 543.375,A -85,B 0,C 180,E1 -27789.306,E2 -27789.306} C_VEL
LIN {X 0,Y 77.14,Z 545.839,A -85,B 0,C 180,E1 -27799.502,E2 -27799.502} C_VEL
LIN {X 0,Y 76.735,Z 546.437,A -85,B 0,C 180,E1 -27804.745,E2 -27804.745} C_VEL
LIN {X 0,Y 76.781,Z 546.6,A -85,B 0,C 180,E1 -27810,E2 -27810} C_VEL
LIN {X 0,Y 76.711,Z 546.437,A -85,B 0,C 180,E1 -27815.256,E2 -27815.256} C_VEL
LIN {X 0,Y 77.125,Z 545.838,A -85,B 0,C 180,E1 -27820.501,E2 -27820.501} C_VEL
LIN {X 0,Y 79.55,Z 543.375,A -85,B 0,C 180,E1 -27830.694,E2 -27830.694} C_VEL
LIN {X 0,Y 82.784,Z 540.416,A -85,B 0,C 180,E1 -27837.834,E2 -27837.834} C_VEL
LIN {X 0,Y 87.25,Z 536.425,A -85,B 0,C 180,E1 -27844.321,E2 -27844.321} C_VEL
LIN {X 0,Y 92.711,Z 531.295,A -85,B 0,C 180,E1 -27850.116,E2 -27850.116} C_VEL
LIN {X 0,Y 97.625,Z 526.143,A -85,B 0,C 180,E1 -27854.434,E2 -27854.434} C_VEL
LIN {X 0,Y 102.19,Z 521.087,A -85,B 0,C 180,E1 -27857.672,E2 -27857.672} C_VEL
LIN {X 0,Y 103.222,Z 519.706,A -85,B 0,C 180,E1 -27858.498,E2 -27858.498} C_VEL
LIN {X 0,Y 106.048,Z 513.666,A -85,B 0,C 180,E1 -27862.679,E2 -27862.679} C_VEL
LIN {X 0,Y 108.01,Z 508.54,A -85,B 0,C 180,E1 -27866.081,E2 -27866.081} C_VEL
LIN {X 0,Y 109.136,Z 504.174,A -85,B 0,C 180,E1 -27868.989,E2 -27868.989} C_VEL
LIN {X 0,Y 109.462,Z 500.19,A -85,B 0,C 180,E1 -27872.256,E2 -27872.256} C_VEL
LIN {X 0,Y 109.191,Z 495,A -85,B 0,C 180,E1 -27877.28,E2 -27877.28} C_VEL
LIN {X 0,Y 108.82,Z 491.696,A -85,B 0,C 180,E1 -27881.158,E2 -27881.158} C_VEL
LIN {X 0,Y 108.384,Z 488.916,A -85,B 0,C 180,E1 -27884.965,E2 -27884.965} C_VEL
LIN {X 0,Y 108.059,Z 486.713,A -85,B 0,C 180,E1 -27888.746,E2 -27888.746} C_VEL
LIN {X 0,Y 107.72,Z 483.441,A -85,B 0,C 180,E1 -27899.998,E2 -27899.998} C_VEL
LIN {X 0,Y 107.592,Z 486.271,A -85,B 0,C 180,E1 -27911.299,E2 -27911.299} C_VEL
LIN {X 0,Y 108.367,Z 488.828,A -85,B 0,C 180,E1 -27916.966,E2 -27916.966} C_VEL
LIN {X 0,Y 109.374,Z 492.399,A -85,B 0,C 180,E1 -27922.675,E2 -27922.675} C_VEL
LIN {X 0,Y 110.33,Z 497.25,A -85,B 0,C 180,E1 -27928.536,E2 -27928.536} C_VEL
LIN {X 0,Y 110.94,Z 501.961,A -85,B 0,C 180,E1 -27933.437,E2 -27933.437} C_VEL
LIN {X 0,Y 111.281,Z 506.889,A -85,B 0,C 180,E1 -27938.005,E2 -27938.005} C_VEL
LIN {X 0,Y 111.123,Z 512.411,A -85,B 0,C 180,E1 -27942.846,E2 -27942.846} C_VEL
LIN {X 0,Y 110.397,Z 518.271,A -85,B 0,C 180,E1 -27948.057,E2 -27948.057} C_VEL
LIN {X 0,Y 109.633,Z 524.938,A -85,B 0,C 180,E1 -27954.765,E2 -27954.765} C_VEL
LIN {X 0,Y 110.473,Z 529.964,A -85,B 0,C 180,E1 -27961.192,E2 -27961.192} C_VEL
LIN {X 0,Y 112.238,Z 533.1,A -85,B 0,C 180,E1 -27965.983,E2 -27965.983} C_VEL
LIN {X 0,Y 117.253,Z 536.889,A -85,B 0,C 180,E1 -27973.533,E2 -27973.533} C_VEL
LIN {X 0,Y 122.035,Z 538.735,A -85,B 0,C 180,E1 -27978.236,E2 -27978.236} C_VEL
LIN {X 0,Y 126.106,Z 539.587,A -85,B 0,C 180,E1 -27981.374,E2 -27981.374} C_VEL
LIN {X 0,Y 126.695,Z 539.98,A -85,B 0,C 180,E1 -27982.543,E2 -27982.543} C_VEL
LIN {X 0,Y 125.519,Z 540.702,A -85,B 0,C 180,E1 -27985.969,E2 -27985.969} C_VEL
LIN {X 0,Y 126.295,Z 540.841,A -85,B 0,C 180,E1 -27986.942,E2 -27986.942} C_VEL
LIN {X 0,Y 132.206,Z 540.8,A -85,B 0,C 180,E1 -27990,E2 -27990} C_VEL
LIN {X 0,Y 126.049,Z 540.824,A -85,B 0,C 180,E1 -27993.196,E2 -27993.196} C_VEL
LIN {X 0,Y 120.311,Z 540.408,A -85,B 0,C 180,E1 -27996.771,E2 -27996.771} C_VEL
LIN {X 0,Y 111.32,Z 538.321,A -85,B 0,C 180,E1 -28004.627,E2 -28004.627} C_VEL
LIN {X 0,Y 107.901,Z 536.695,A -85,B 0,C 180,E1 -28009.006,E2 -28009.006} C_VEL
LIN {X 0,Y 104.4,Z 533.363,A -85,B 0,C 180,E1 -28015.912,E2 -28015.912} C_VEL
LIN {X 0,Y 102.96,Z 528.838,A -85,B 0,C 180,E1 -28023.097,E2 -28023.097} C_VEL
LIN {X 0,Y 103.326,Z 523.416,A -85,B 0,C 180,E1 -28029.838,E2 -28029.838} C_VEL
LIN {X 0,Y 104.405,Z 518.498,A -85,B 0,C 180,E1 -28034.974,E2 -28034.974} C_VEL
LIN {X 0,Y 105.2,Z 512.805,A -85,B 0,C 180,E1 -28040.608,E2 -28040.608} C_VEL
LIN {X 0,Y 105.378,Z 508.4,A -85,B 0,C 180,E1 -28044.969,E2 -28044.969} C_VEL
LIN {X 0,Y 105.232,Z 503.533,A -85,B 0,C 180,E1 -28050.249,E2 -28050.249} C_VEL
LIN {X 0,Y 104.888,Z 499.839,A -85,B 0,C 180,E1 -28054.856,E2 -28054.856} C_VEL
LIN {X 0,Y 104.582,Z 497.316,A -85,B 0,C 180,E1 -28058.311,E2 -28058.311} C_VEL
LIN {X 0,Y 103.896,Z 493.947,A -85,B 0,C 180,E1 -28064.304,E2 -28064.304} C_VEL
LIN {X 0,Y 103.582,Z 492.348,A -85,B 0,C 180,E1 -28068.258,E2 -28068.258} C_VEL
LIN {X 0,Y 103.38,Z 490.292,A -85,B 0,C 180,E1 -28076.104,E2 -28076.104} C_VEL
LIN {X 0,Y 103.792,Z 489.488,A -85,B 0,C 180,E1 -28080.002,E2 -28080.002} C_VEL
LIN {X 0,Y 103.664,Z 491.544,A -85,B 0,C 180,E1 -28087.795,E2 -28087.795} C_VEL
LIN {X 0,Y 103.999,Z 492.967,A -85,B 0,C 180,E1 -28091.699,E2 -28091.699} C_VEL
LIN {X 0,Y 104.153,Z 495.166,A -85,B 0,C 180,E1 -28095.661,E2 -28095.661} C_VEL
LIN {X 0,Y 104.265,Z 498.094,A -85,B 0,C 180,E1 -28099.698,E2 -28099.698} C_VEL
LIN {X 0,Y 104.326,Z 501.728,A -85,B 0,C 180,E1 -28103.843,E2 -28103.843} C_VEL
LIN {X 0,Y 103.932,Z 506.144,A -85,B 0,C 180,E1 -28108.254,E2 -28108.254} C_VEL
LIN {X 0,Y 103.469,Z 508.248,A -85,B 0,C 180,E1 -28109.921,E2 -28109.921} C_VEL
LIN {X 0,Y 100.79,Z 514.714,A -85,B 0,C 180,E1 -28114.58,E2 -28114.58} C_VEL
LIN {X 0,Y 97.469,Z 520.887,A -85,B 0,C 180,E1 -28119.185,E2 -28119.185} C_VEL
LIN {X 0,Y 90.536,Z 528.141,A -85,B 0,C 180,E1 -28124.108,E2 -28124.108} C_VEL
LIN {X 0,Y 85.337,Z 533.013,A -85,B 0,C 180,E1 -28128.789,E2 -28128.789} C_VEL
LIN {X 0,Y 79.721,Z 537.759,A -85,B 0,C 180,E1 -28135.04,E2 -28135.04} C_VEL
LIN {X 0,Y 75.151,Z 541.369,A -85,B 0,C 180,E1 -28142.122,E2 -28142.122} C_VEL
LIN {X 0,Y 72.918,Z 543.177,A -85,B 0,C 180,E1 -28147.324,E2 -28147.324} C_VEL
LIN {X 0,Y 70.158,Z 545.641,A -85,B 0,C 180,E1 -28158.443,E2 -28158.443} C_VEL
LIN {X 0,Y 69.648,Z 546.24,A -85,B 0,C 180,E1 -28164.209,E2 -28164.209} C_VEL
LIN {X 0,Y 69.701,Z 546.403,A -85,B 0,C 180,E1 -28170,E2 -28170} C_VEL
LIN {X 0,Y 69.624,Z 546.239,A -85,B 0,C 180,E1 -28175.793,E2 -28175.793} C_VEL
LIN {X 0,Y 70.146,Z 545.641,A -85,B 0,C 180,E1 -28181.559,E2 -28181.559} C_VEL
LIN {X 0,Y 72.918,Z 543.177,A -85,B 0,C 180,E1 -28192.676,E2 -28192.676} C_VEL
LIN {X 0,Y 76.558,Z 540.218,A -85,B 0,C 180,E1 -28200.324,E2 -28200.324} C_VEL
LIN {X 0,Y 81.451,Z 536.226,A -85,B 0,C 180,E1 -28207.155,E2 -28207.155} C_VEL
LIN {X 0,Y 87.236,Z 531.215,A -85,B 0,C 180,E1 -28213.022,E2 -28213.022} C_VEL
LIN {X 0,Y 92.765,Z 525.829,A -85,B 0,C 180,E1 -28217.617,E2 -28217.617} C_VEL
LIN {X 0,Y 97.462,Z 520.886,A -85,B 0,C 180,E1 -28220.82,E2 -28220.82} C_VEL
LIN {X 0,Y 100.772,Z 514.734,A -85,B 0,C 180,E1 -28225.413,E2 -28225.413} C_VEL
LIN {X 0,Y 102.785,Z 510.121,A -85,B 0,C 180,E1 -28228.724,E2 -28228.724} C_VEL
LIN {X 0,Y 103.913,Z 506.167,A -85,B 0,C 180,E1 -28231.74,E2 -28231.74} C_VEL
LIN {X 0,Y 104.324,Z 501.729,A -85,B 0,C 180,E1 -28236.157,E2 -28236.157} C_VEL
LIN {X 0,Y 104.246,Z 497.785,A -85,B 0,C 180,E1 -28240.703,E2 -28240.703} C_VEL
LIN {X 0,Y 104.167,Z 495.148,A -85,B 0,C 180,E1 -28244.341,E2 -28244.341} C_VEL
LIN {X 0,Y 104.012,Z 492.949,A -85,B 0,C 180,E1 -28248.303,E2 -28248.303} C_VEL
LIN {X 0,Y 103.676,Z 491.526,A -85,B 0,C 180,E1 -28252.206,E2 -28252.206} C_VEL
LIN {X 0,Y 103.807,Z 489.466,A -85,B 0,C 180,E1 -28259.998,E2 -28259.998} C_VEL
LIN {X 0,Y 103.369,Z 491.202,A -85,B 0,C 180,E1 -28267.813,E2 -28267.813} C_VEL
LIN {X 0,Y 103.574,Z 492.358,A -85,B 0,C 180,E1 -28271.743,E2 -28271.743} C_VEL
LIN {X 0,Y 103.89,Z 493.955,A -85,B 0,C 180,E1 -28275.697,E2 -28275.697} C_VEL
LIN {X 0,Y 104.58,Z 497.319,A -85,B 0,C 180,E1 -28281.689,E2 -28281.689} C_VEL
LIN {X 0,Y 105.029,Z 500.894,A -85,B 0,C 180,E1 -28286.592,E2 -28286.592} C_VEL
LIN {X 0,Y 105.352,Z 504.631,A -85,B 0,C 180,E1 -28291.002,E2 -28291.002} C_VEL
LIN {X 0,Y 105.375,Z 510.174,A -85,B 0,C 180,E1 -28296.886,E2 -28296.886} C_VEL
LIN {X 0,Y 104.863,Z 515.449,A -85,B 0,C 180,E1 -28302.08,E2 -28302.08} C_VEL
LIN {X 0,Y 104.142,Z 519.707,A -85,B 0,C 180,E1 -28306.235,E2 -28306.235} C_VEL
LIN {X 0,Y 102.883,Z 526.56,A -85,B 0,C 180,E1 -28313.923,E2 -28313.923} C_VEL
LIN {X 0,Y 103.208,Z 530.419,A -85,B 0,C 180,E1 -28319.289,E2 -28319.289} C_VEL
LIN {X 0,Y 104.415,Z 533.364,A -85,B 0,C 180,E1 -28324.095,E2 -28324.095} C_VEL
LIN {X 0,Y 107.859,Z 536.696,A -85,B 0,C 180,E1 -28330.987,E2 -28330.987} C_VEL
LIN {X 0,Y 114.638,Z 539.358,A -85,B 0,C 180,E1 -28338.773,E2 -28338.773} C_VEL
LIN {X 0,Y 120.384,Z 540.416,A -85,B 0,C 180,E1 -28343.295,E2 -28343.295} C_VEL
LIN {X 0,Y 126.295,Z 540.841,A -85,B 0,C 180,E1 -28346.942,E2 -28346.942} C_VEL
LIN {X 0,Y 126.861,Z 540.946,A -85,B 0,C 180,E1 -28347.893,E2 -28347.893} C_VEL
LIN {X 0,Y 126.03,Z 541.031,A -85,B 0,C 180,E1 -28349.177,E2 -28349.177} C_VEL
LIN {X 0,Y 124.217,Z 541.089,A -85,B 0,C 180,E1 -28350.402,E2 -28350.402} C_VEL
LIN {X 0,Y 114.925,Z 540.963,A -85,B 0,C 180,E1 -28354.586,E2 -28354.586} C_VEL
LIN {X 0,Y 113.911,Z 540.891,A -85,B 0,C 180,E1 -28355.227,E2 -28355.227} C_VEL
LIN {X 0,Y 106.52,Z 539.787,A -85,B 0,C 180,E1 -28361.416,E2 -28361.416} C_VEL
LIN {X 0,Y 102.434,Z 538.479,A -85,B 0,C 180,E1 -28366.158,E2 -28366.158} C_VEL
LIN {X 0,Y 98.767,Z 536.236,A -85,B 0,C 180,E1 -28372.331,E2 -28372.331} C_VEL
LIN {X 0,Y 96.347,Z 532.126,A -85,B 0,C 180,E1 -28380.704,E2 -28380.704} C_VEL
LIN {X 0,Y 96.287,Z 527.233,A -85,B 0,C 180,E1 -28388.343,E2 -28388.343} C_VEL
LIN {X 0,Y 97.937,Z 521.051,A -85,B 0,C 180,E1 -28395.856,E2 -28395.856} C_VEL
LIN {X 0,Y 98.834,Z 517.113,A -85,B 0,C 180,E1 -28400.212,E2 -28400.212} C_VEL
LIN {X 0,Y 99.51,Z 512.376,A -85,B 0,C 180,E1 -28405.6,E2 -28405.6} C_VEL
LIN {X 0,Y 99.732,Z 508.282,A -85,B 0,C 180,E1 -28410.446,E2 -28410.446} C_VEL
LIN {X 0,Y 99.615,Z 503.88,A -85,B 0,C 180,E1 -28416.512,E2 -28416.512} C_VEL
LIN {X 0,Y 99.472,Z 501.166,A -85,B 0,C 180,E1 -28420.979,E2 -28420.979} C_VEL
LIN {X 0,Y 99.362,Z 499.909,A -85,B 0,C 180,E1 -28423.568,E2 -28423.568} C_VEL
LIN {X 0,Y 99.146,Z 498.189,A -85,B 0,C 180,E1 -28427.724,E2 -28427.724} C_VEL
LIN {X 0,Y 99.099,Z 496.041,A -85,B 0,C 180,E1 -28435.936,E2 -28435.936} C_VEL
LIN {X 0,Y 99.577,Z 495.299,A -85,B 0,C 180,E1 -28440.002,E2 -28440.002} C_VEL
LIN {X 0,Y 99.296,Z 497.341,A -85,B 0,C 180,E1 -28448.14,E2 -28448.14} C_VEL
LIN {X 0,Y 99.465,Z 498.941,A -85,B 0,C 180,E1 -28452.24,E2 -28452.24} C_VEL
LIN {X 0,Y 99.439,Z 501.383,A -85,B 0,C 180,E1 -28456.424,E2 -28456.424} C_VEL
LIN {X 0,Y 99.183,Z 504.448,A -85,B 0,C 180,E1 -28460.752,E2 -28460.752} C_VEL
LIN {X 0,Y 98.794,Z 508.35,A -85,B 0,C 180,E1 -28465.269,E2 -28465.269} C_VEL
LIN {X 0,Y 98.231,Z 510.399,A -85,B 0,C 180,E1 -28467.292,E2 -28467.292} C_VEL
LIN {X 0,Y 96.31,Z 514.667,A -85,B 0,C 180,E1 -28470.72,E2 -28470.72} C_VEL
LIN {X 0,Y 92.78,Z 520.672,A -85,B 0,C 180,E1 -28475.484,E2 -28475.484} C_VEL
LIN {X 0,Y 91.88,Z 522.066,A -85,B 0,C 180,E1 -28476.569,E2 -28476.569} C_VEL
LIN {X 0,Y 83.849,Z 529.551,A -85,B 0,C 180,E1 -28482.112,E2 -28482.112} C_VEL
LIN {X 0,Y 77.944,Z 534.475,A -85,B 0,C 180,E1 -28487.45,E2 -28487.45} C_VEL
LIN {X 0,Y 72.185,Z 538.802,A -85,B 0,C 180,E1 -28494.257,E2 -28494.257} C_VEL
LIN {X 0,Y 68.932,Z 541.172,A -85,B 0,C 180,E1 -28499.352,E2 -28499.352} C_VEL
LIN {X 0,Y 66.377,Z 542.978,A -85,B 0,C 180,E1 -28504.943,E2 -28504.943} C_VEL
LIN {X 0,Y 63.192,Z 545.443,A -85,B 0,C 180,E1 -28517.148,E2 -28517.148} C_VEL
LIN {X 0,Y 62.578,Z 546.042,A -85,B 0,C 180,E1 -28523.552,E2 -28523.552} C_VEL
LIN {X 0,Y 62.611,Z 546.207,A -85,B 0,C 180,E1 -28530,E2 -28530} C_VEL
LIN {X 0,Y 62.559,Z 546.042,A -85,B 0,C 180,E1 -28536.45,E2 -28536.45} C_VEL
LIN {X 0,Y 63.183,Z 545.443,A -85,B 0,C 180,E1 -28542.854,E2 -28542.854} C_VEL
LIN {X 0,Y 66.377,Z 542.978,A -85,B 0,C 180,E1 -28555.056,E2 -28555.056} C_VEL
LIN {X 0,Y 70.506,Z 540.021,A -85,B 0,C 180,E1 -28563.245,E2 -28563.245} C_VEL
LIN {X 0,Y 75.889,Z 536.028,A -85,B 0,C 180,E1 -28570.41,E2 -28570.41} C_VEL
LIN {X 0,Y 81.391,Z 531.686,A -85,B 0,C 180,E1 -28575.743,E2 -28575.743} C_VEL
LIN {X 0,Y 86.913,Z 526.788,A -85,B 0,C 180,E1 -28580.19,E2 -28580.19} C_VEL
LIN {X 0,Y 91.857,Z 522.065,A -85,B 0,C 180,E1 -28583.45,E2 -28583.45} C_VEL
LIN {X 0,Y 95.661,Z 515.95,A -85,B 0,C 180,E1 -28588.333,E2 -28588.333} C_VEL
LIN {X 0,Y 97.503,Z 512.12,A -85,B 0,C 180,E1 -28591.253,E2 -28591.253} C_VEL
LIN {X 0,Y 98.566,Z 509.344,A -85,B 0,C 180,E1 -28593.738,E2 -28593.738} C_VEL
LIN {X 0,Y 99.037,Z 506.043,A -85,B 0,C 180,E1 -28597.294,E2 -28597.294} C_VEL
LIN {X 0,Y 99.3,Z 503.145,A -85,B 0,C 180,E1 -28600.972,E2 -28600.972} C_VEL
LIN {X 0,Y 99.512,Z 500.044,A -85,B 0,C 180,E1 -28605.687,E2 -28605.687} C_VEL
LIN {X 0,Y 99.467,Z 498.938,A -85,B 0,C 180,E1 -28607.76,E2 -28607.76} C_VEL
LIN {X 0,Y 99.305,Z 497.202,A -85,B 0,C 180,E1 -28612.217,E2 -28612.217} C_VEL
LIN {X 0,Y 99.599,Z 495.271,A -85,B 0,C 180,E1 -28619.998,E2 -28619.998} C_VEL
LIN {X 0,Y 98.992,Z 496.954,A -85,B 0,C 180,E1 -28628.161,E2 -28628.161} C_VEL
LIN {X 0,Y 99.143,Z 498.193,A -85,B 0,C 180,E1 -28632.276,E2 -28632.276} C_VEL
LIN {X 0,Y 99.358,Z 499.914,A -85,B 0,C 180,E1 -28636.433,E2 -28636.433} C_VEL
LIN {X 0,Y 99.583,Z 502.03,A -85,B 0,C 180,E1 -28640.661,E2 -28640.661} C_VEL
LIN {X 0,Y 99.739,Z 504.872,A -85,B 0,C 180,E1 -28645.008,E2 -28645.008} C_VEL
LIN {X 0,Y 99.767,Z 508.244,A -85,B 0,C 180,E1 -28649.542,E2 -28649.542} C_VEL
LIN {X 0,Y 99.441,Z 513.597,A -85,B 0,C 180,E1 -28655.821,E2 -28655.821} C_VEL
LIN {X 0,Y 98.504,Z 519.067,A -85,B 0,C 180,E1 -28661.882,E2 -28661.882} C_VEL
LIN {X 0,Y 96.699,Z 525.393,A -85,B 0,C 180,E1 -28669.149,E2 -28669.149} C_VEL
LIN {X 0,Y 96.082,Z 530.652,A -85,B 0,C 180,E1 -28676.73,E2 -28676.73} C_VEL
LIN {X 0,Y 97.478,Z 534.737,A -85,B 0,C 180,E1 -28684.369,E2 -28684.369} C_VEL
LIN {X 0,Y 99.606,Z 536.939,A -85,B 0,C 180,E1 -28689.342,E2 -28689.342} C_VEL
LIN {X 0,Y 102.572,Z 538.572,A -85,B 0,C 180,E1 -28694.094,E2 -28694.094} C_VEL
LIN {X 0,Y 111.151,Z 540.674,A -85,B 0,C 180,E1 -28702.735,E2 -28702.735} C_VEL
LIN {X 0,Y 120.878,Z 541.115,A -85,B 0,C 180,E1 -28709.046,E2 -28709.046} C_VEL
LIN {X 0,Y 122.667,Z 541.065,A -85,B 0,C 180,E1 -28710,E2 -28710} C_VEL
LIN {X 0,Y 113.911,Z 540.891,A -85,B 0,C 180,E1 -28715.227,E2 -28715.227} C_VEL
LIN {X 0,Y 110.039,Z 540.678,A -85,B 0,C 180,E1 -28717.516,E2 -28717.516} C_VEL
LIN {X 0,Y 97.328,Z 539.587,A -85,B 0,C 180,E1 -28724.42,E2 -28724.42} C_VEL
LIN {X 0,Y 94.226,Z 538.815,A -85,B 0,C 180,E1 -28727.369,E2 -28727.369} C_VEL
LIN {X 0,Y 93.502,Z 538.469,A -85,B 0,C 180,E1 -28728.461,E2 -28728.461} C_VEL
LIN {X 0,Y 90.502,Z 536.115,A -85,B 0,C 180,E1 -28735.281,E2 -28735.281} C_VEL
LIN {X 0,Y 89.242,Z 532.359,A -85,B 0,C 180,E1 -28743.453,E2 -28743.453} C_VEL
LIN {X 0,Y 89.549,Z 529.297,A -85,B 0,C 180,E1 -28748.891,E2 -28748.891} C_VEL
LIN {X 0,Y 91.259,Z 524.128,A -85,B 0,C 180,E1 -28756.127,E2 -28756.127} C_VEL
LIN {X 0,Y 92.661,Z 519.871,A -85,B 0,C 180,E1 -28761.503,E2 -28761.503} C_VEL
LIN {X 0,Y 93.405,Z 516.353,A -85,B 0,C 180,E1 -28765.858,E2 -28765.858} C_VEL
LIN {X 0,Y 94.028,Z 512.594,A -85,B 0,C 180,E1 -28770.936,E2 -28770.936} C_VEL
LIN {X 0,Y 94.293,Z 508.836,A -85,B 0,C 180,E1 -28776.551,E2 -28776.551} C_VEL
LIN {X 0,Y 94.484,Z 506.621,A -85,B 0,C 180,E1 -28780.447,E2 -28780.447} C_VEL
LIN {X 0,Y 94.313,Z 503.782,A -85,B 0,C 180,E1 -28787.085,E2 -28787.085} C_VEL
LIN {X 0,Y 94.33,Z 502.507,A -85,B 0,C 180,E1 -28791.433,E2 -28791.433} C_VEL
LIN {X 0,Y 95.102,Z 500.91,A -85,B 0,C 180,E1 -28800.002,E2 -28800.002} C_VEL
LIN {X 0,Y 94.618,Z 502.97,A -85,B 0,C 180,E1 -28808.546,E2 -28808.546} C_VEL
LIN {X 0,Y 94.575,Z 504.661,A -85,B 0,C 180,E1 -28812.884,E2 -28812.884} C_VEL
LIN {X 0,Y 94.212,Z 507.334,A -85,B 0,C 180,E1 -28817.363,E2 -28817.363} C_VEL
LIN {X 0,Y 93.575,Z 510.652,A -85,B 0,C 180,E1 -28822.059,E2 -28822.059} C_VEL
LIN {X 0,Y 92.637,Z 513.646,A -85,B 0,C 180,E1 -28825.488,E2 -28825.488} C_VEL
LIN {X 0,Y 90.74,Z 517.086,A -85,B 0,C 180,E1 -28828.463,E2 -28828.463} C_VEL
LIN {X 0,Y 87.501,Z 521.852,A -85,B 0,C 180,E1 -28832.506,E2 -28832.506} C_VEL
LIN {X 0,Y 86.489,Z 523.123,A -85,B 0,C 180,E1 -28833.604,E2 -28833.604} C_VEL
LIN {X 0,Y 78.561,Z 529.874,A -85,B 0,C 180,E1 -28838.775,E2 -28838.775} C_VEL
LIN {X 0,Y 72.862,Z 534.277,A -85,B 0,C 180,E1 -28843.664,E2 -28843.664} C_VEL
LIN {X 0,Y 66.537,Z 538.605,A -85,B 0,C 180,E1 -28850.674,E2 -28850.674} C_VEL
LIN {X 0,Y 62.912,Z 540.974,A -85,B 0,C 180,E1 -28856.045,E2 -28856.045} C_VEL
LIN {X 0,Y 57.774,Z 544.177,A -85,B 0,C 180,E1 -28868.597,E2 -28868.597} C_VEL
LIN {X 0,Y 56.279,Z 545.246,A -85,B 0,C 180,E1 -28875.537,E2 -28875.537} C_VEL
LIN {X 0,Y 55.531,Z 545.846,A -85,B 0,C 180,E1 -28882.729,E2 -28882.729} C_VEL
LIN {X 0,Y 55.509,Z 546.01,A -85,B 0,C 180,E1 -28890,E2 -28890} C_VEL
LIN {X 0,Y 55.517,Z 545.845,A -85,B 0,C 180,E1 -28897.273,E2 -28897.273} C_VEL
LIN {X 0,Y 56.272,Z 545.246,A -85,B 0,C 180,E1 -28904.465,E2 -28904.465} C_VEL
LIN {X 0,Y 59.978,Z 542.78,A -85,B 0,C 180,E1 -28917.95,E2 -28917.95} C_VEL
LIN {X 0,Y 64.675,Z 539.823,A -85,B 0,C 180,E1 -28926.702,E2 -28926.702} C_VEL
LIN {X 0,Y 70.615,Z 535.831,A -85,B 0,C 180,E1 -28934.16,E2 -28934.16} C_VEL
LIN {X 0,Y 77.299,Z 530.869,A -85,B 0,C 180,E1 -28940.242,E2 -28940.242} C_VEL
LIN {X 0,Y 83.812,Z 525.433,A -85,B 0,C 180,E1 -28944.842,E2 -28944.842} C_VEL
LIN {X 0,Y 86.452,Z 523.121,A -85,B 0,C 180,E1 -28946.433,E2 -28946.433} C_VEL
LIN {X 0,Y 89.41,Z 519.054,A -85,B 0,C 180,E1 -28949.84,E2 -28949.84} C_VEL
LIN {X 0,Y 92.311,Z 514.32,A -85,B 0,C 180,E1 -28953.919,E2 -28953.919} C_VEL
LIN {X 0,Y 93.247,Z 511.951,A -85,B 0,C 180,E1 -28956.306,E2 -28956.306} C_VEL
LIN {X 0,Y 93.977,Z 508.913,A -85,B 0,C 180,E1 -28960.332,E2 -28960.332} C_VEL
LIN {X 0,Y 94.455,Z 505.647,A -85,B 0,C 180,E1 -28965.296,E2 -28965.296} C_VEL
LIN {X 0,Y 94.578,Z 504.658,A -85,B 0,C 180,E1 -28967.117,E2 -28967.117} C_VEL
LIN {X 0,Y 94.625,Z 502.963,A -85,B 0,C 180,E1 -28971.455,E2 -28971.455} C_VEL
LIN {X 0,Y 95.129,Z 500.88,A -85,B 0,C 180,E1 -28979.998,E2 -28979.998} C_VEL
LIN {X 0,Y 94.332,Z 502.504,A -85,B 0,C 180,E1 -28988.567,E2 -28988.567} C_VEL
LIN {X 0,Y 94.312,Z 504.333,A -85,B 0,C 180,E1 -28994.369,E2 -28994.369} C_VEL
LIN {X 0,Y 94.483,Z 506.622,A -85,B 0,C 180,E1 -28999.553,E2 -28999.553} C_VEL
LIN {X 0,Y 94.336,Z 508.833,A -85,B 0,C 180,E1 -29003.508,E2 -29003.508} C_VEL
LIN {X 0,Y 94.048,Z 512.573,A -85,B 0,C 180,E1 -29009.057,E2 -29009.057} C_VEL
LIN {X 0,Y 93.459,Z 516.35,A -85,B 0,C 180,E1 -29014.191,E2 -29014.191} C_VEL
LIN {X 0,Y 92.67,Z 519.863,A -85,B 0,C 180,E1 -29018.492,E2 -29018.492} C_VEL
LIN {X 0,Y 91.253,Z 524.134,A -85,B 0,C 180,E1 -29023.877,E2 -29023.877} C_VEL
LIN {X 0,Y 89.457,Z 529.737,A -85,B 0,C 180,E1 -29031.774,E2 -29031.774} C_VEL
LIN {X 0,Y 89.504,Z 534.015,A -85,B 0,C 180,E1 -29039.734,E2 -29039.734} C_VEL
LIN {X 0,Y 91.485,Z 537.182,A -85,B 0,C 180,E1 -29047.412,E2 -29047.412} C_VEL
LIN {X 0,Y 95.014,Z 539.274,A -85,B 0,C 180,E1 -29054.057,E2 -29054.057} C_VEL
LIN {X 0,Y 102.041,Z 540.929,A -85,B 0,C 180,E1 -29062.083,E2 -29062.083} C_VEL
LIN {X 0,Y 107.182,Z 541.349,A -85,B 0,C 180,E1 -29066.24,E2 -29066.24} C_VEL
LIN {X 0,Y 113.152,Z 541.329,A -85,B 0,C 180,E1 -29070,E2 -29070} C_VEL
LIN {X 0,Y 105.787,Z 541.24,A -85,B 0,C 180,E1 -29074.799,E2 -29074.799} C_VEL
LIN {X 0,Y 99.906,Z 540.578,A -85,B 0,C 180,E1 -29080.003,E2 -29080.003} C_VEL
LIN {X 0,Y 94.131,Z 538.817,A -85,B 0,C 180,E1 -29087.376,E2 -29087.376} C_VEL
LIN {X 0,Y 93.502,Z 538.469,A -85,B 0,C 180,E1 -29088.461,E2 -29088.461} C_VEL
LIN {X 0,Y 91.191,Z 537.521,A -85,B 0,C 180,E1 -29091.787,E2 -29091.787} C_VEL
LIN {X 0,Y 83.504,Z 534.43,A -85,B 0,C 180,E1 -29102.162,E2 -29102.162} C_VEL
LIN {X 0,Y 82.478,Z 532.893,A -85,B 0,C 180,E1 -29106.003,E2 -29106.003} C_VEL
LIN {X 0,Y 82.494,Z 532.259,A -85,B 0,C 180,E1 -29107.29,E2 -29107.29} C_VEL
LIN {X 0,Y 84.142,Z 527.683,A -85,B 0,C 180,E1 -29115.231,E2 -29115.231} C_VEL
LIN {X 0,Y 85.882,Z 523.747,A -85,B 0,C 180,E1 -29121.019,E2 -29121.019} C_VEL
LIN {X 0,Y 87.397,Z 519.527,A -85,B 0,C 180,E1 -29127.129,E2 -29127.129} C_VEL
LIN {X 0,Y 88.339,Z 515.347,A -85,B 0,C 180,E1 -29133.502,E2 -29133.502} C_VEL
LIN {X 0,Y 88.908,Z 512.146,A -85,B 0,C 180,E1 -29139.168,E2 -29139.168} C_VEL
LIN {X 0,Y 89.091,Z 510.911,A -85,B 0,C 180,E1 -29141.609,E2 -29141.609} C_VEL
LIN {X 0,Y 89.217,Z 509.122,A -85,B 0,C 180,E1 -29146.333,E2 -29146.333} C_VEL
LIN {X 0,Y 89.388,Z 507.853,A -85,B 0,C 180,E1 -29150.955,E2 -29150.955} C_VEL
LIN {X 0,Y 89.692,Z 506.905,A -85,B 0,C 180,E1 -29155.508,E2 -29155.508} C_VEL
LIN {X 0,Y 90.236,Z 506.208,A -85,B 0,C 180,E1 -29160.002,E2 -29160.002} C_VEL
LIN {X 0,Y 89.628,Z 508.403,A -85,B 0,C 180,E1 -29169.025,E2 -29169.025} C_VEL
LIN {X 0,Y 89.277,Z 510.238,A -85,B 0,C 180,E1 -29173.663,E2 -29173.663} C_VEL
LIN {X 0,Y 88.485,Z 513.063,A -85,B 0,C 180,E1 -29178.527,E2 -29178.527} C_VEL
LIN {X 0,Y 87.584,Z 515.863,A -85,B 0,C 180,E1 -29182.408,E2 -29182.408} C_VEL
LIN {X 0,Y 85.61,Z 518.828,A -85,B 0,C 180,E1 -29185.444,E2 -29185.444} C_VEL
LIN {X 0,Y 82.483,Z 522.91,A -85,B 0,C 180,E1 -29189.151,E2 -29189.151} C_VEL
LIN {X 0,Y 81.341,Z 524.081,A -85,B 0,C 180,E1 -29190.232,E2 -29190.232} C_VEL
LIN {X 0,Y 75.839,Z 528.584,A -85,B 0,C 180,E1 -29193.487,E2 -29193.487} C_VEL
LIN {X 0,Y 68.145,Z 534.08,A -85,B 0,C 180,E1 -29199.332,E2 -29199.332} C_VEL
LIN {X 0,Y 61.197,Z 538.407,A -85,B 0,C 180,E1 -29206.446,E2 -29206.446} C_VEL
LIN {X 0,Y 57.151,Z 540.777,A -85,B 0,C 180,E1 -29212.059,E2 -29212.059} C_VEL
LIN {X 0,Y 53.771,Z 542.582,A -85,B 0,C 180,E1 -29218.48,E2 -29218.48} C_VEL
LIN {X 0,Y 49.403,Z 545.048,A -85,B 0,C 180,E1 -29233.47,E2 -29233.47} C_VEL
LIN {X 0,Y 48.489,Z 545.648,A -85,B 0,C 180,E1 -29241.666,E2 -29241.666} C_VEL
LIN {X 0,Y 48.427,Z 545.813,A -85,B 0,C 180,E1 -29250,E2 -29250} C_VEL
LIN {X 0,Y 48.477,Z 545.648,A -85,B 0,C 180,E1 -29258.336,E2 -29258.336} C_VEL
LIN {X 0,Y 49.396,Z 545.048,A -85,B 0,C 180,E1 -29266.532,E2 -29266.532} C_VEL
LIN {X 0,Y 53.771,Z 542.582,A -85,B 0,C 180,E1 -29281.52,E2 -29281.52} C_VEL
LIN {X 0,Y 59.105,Z 539.625,A -85,B 0,C 180,E1 -29290.842,E2 -29290.842} C_VEL
LIN {X 0,Y 65.694,Z 535.633,A -85,B 0,C 180,E1 -29298.49,E2 -29298.49} C_VEL
LIN {X 0,Y 72.237,Z 531.186,A -85,B 0,C 180,E1 -29304.051,E2 -29304.051} C_VEL
LIN {X 0,Y 79.915,Z 525.235,A -85,B 0,C 180,E1 -29309.029,E2 -29309.029} C_VEL
LIN {X 0,Y 81.312,Z 524.079,A -85,B 0,C 180,E1 -29309.804,E2 -29309.804} C_VEL
LIN {X 0,Y 83.533,Z 521.634,A -85,B 0,C 180,E1 -29312.054,E2 -29312.054} C_VEL
LIN {X 0,Y 86.76,Z 517.21,A -85,B 0,C 180,E1 -29316.105,E2 -29316.105} C_VEL
LIN {X 0,Y 87.579,Z 515.868,A -85,B 0,C 180,E1 -29317.591,E2 -29317.591} C_VEL
LIN {X 0,Y 88.606,Z 512.636,A -85,B 0,C 180,E1 -29322.135,E2 -29322.135} C_VEL
LIN {X 0,Y 89.278,Z 510.236,A -85,B 0,C 180,E1 -29326.337,E2 -29326.337} C_VEL
LIN {X 0,Y 89.635,Z 508.396,A -85,B 0,C 180,E1 -29330.975,E2 -29330.975} C_VEL
LIN {X 0,Y 89.841,Z 507.134,A -85,B 0,C 180,E1 -29335.511,E2 -29335.511} C_VEL
LIN {X 0,Y 90.28,Z 506.16,A -85,B 0,C 180,E1 -29339.998,E2 -29339.998} C_VEL
LIN {X 0,Y 89.393,Z 507.848,A -85,B 0,C 180,E1 -29349.044,E2 -29349.044} C_VEL
LIN {X 0,Y 89.214,Z 509.125,A -85,B 0,C 180,E1 -29353.667,E2 -29353.667} C_VEL
LIN {X 0,Y 89.077,Z 511.086,A -85,B 0,C 180,E1 -29358.782,E2 -29358.782} C_VEL
LIN {X 0,Y 88.765,Z 513.497,A -85,B 0,C 180,E1 -29363.318,E2 -29363.318} C_VEL
LIN {X 0,Y 88.076,Z 516.636,A -85,B 0,C 180,E1 -29368.631,E2 -29368.631} C_VEL
LIN {X 0,Y 87.443,Z 519.485,A -85,B 0,C 180,E1 -29372.85,E2 -29372.85} C_VEL
LIN {X 0,Y 85.907,Z 523.746,A -85,B 0,C 180,E1 -29379.001,E2 -29379.001} C_VEL
LIN {X 0,Y 85.008,Z 525.847,A -85,B 0,C 180,E1 -29381.922,E2 -29381.922} C_VEL
LIN {X 0,Y 82.874,Z 530.756,A -85,B 0,C 180,E1 -29389.746,E2 -29389.746} C_VEL
LIN {X 0,Y 82.448,Z 534.9,A -85,B 0,C 180,E1 -29398.47,E2 -29398.47} C_VEL
LIN {X 0,Y 84.11,Z 537.888,A -85,B 0,C 180,E1 -29406.793,E2 -29406.793} C_VEL
LIN {X 0,Y 88.883,Z 540.289,A -85,B 0,C 180,E1 -29416.278,E2 -29416.278} C_VEL
LIN {X 0,Y 93.008,Z 541.182,A -85,B 0,C 180,E1 -29421.308,E2 -29421.308} C_VEL
LIN {X 0,Y 98.584,Z 541.653,A -85,B 0,C 180,E1 -29426.382,E2 -29426.382} C_VEL
LIN {X 0,Y 103.711,Z 541.591,A -85,B 0,C 180,E1 -29430,E2 -29430} C_VEL
LIN {X 0,Y 98.021,Z 541.604,A -85,B 0,C 180,E1 -29434.111,E2 -29434.111} C_VEL
LIN {X 0,Y 92.556,Z 541.132,A -85,B 0,C 180,E1 -29439.221,E2 -29439.221} C_VEL
LIN {X 0,Y 85.767,Z 539.061,A -85,B 0,C 180,E1 -29449.133,E2 -29449.133} C_VEL
LIN {X 0,Y 83.562,Z 537.422,A -85,B 0,C 180,E1 -29454.867,E2 -29454.867} C_VEL
LIN {X 0,Y 82.369,Z 534.001,A -85,B 0,C 180,E1 -29463.775,E2 -29463.775} C_VEL
LIN {X 0,Y 82.494,Z 532.259,A -85,B 0,C 180,E1 -29467.29,E2 -29467.29} C_VEL
LIN {X 0,Y 82.434,Z 530.463,A -85,B 0,C 180,E1 -29471.198,E2 -29471.198} C_VEL
LIN {X 0,Y 81.335,Z 527.579,A -85,B 0,C 180,E1 -29477.814,E2 -29477.814} C_VEL
LIN {X 0,Y 80.735,Z 523.936,A -85,B 0,C 180,E1 -29485.923,E2 -29485.923} C_VEL
LIN {X 0,Y 81.226,Z 522.419,A -85,B 0,C 180,E1 -29488.536,E2 -29488.536} C_VEL
LIN {X 0,Y 82.506,Z 518.903,A -85,B 0,C 180,E1 -29494.795,E2 -29494.795} C_VEL
LIN {X 0,Y 83.318,Z 516.148,A -85,B 0,C 180,E1 -29500.284,E2 -29500.284} C_VEL
LIN {X 0,Y 83.763,Z 514.271,A -85,B 0,C 180,E1 -29505.424,E2 -29505.424} C_VEL
LIN {X 0,Y 84.03,Z 512.864,A -85,B 0,C 180,E1 -29510.373,E2 -29510.373} C_VEL
LIN {X 0,Y 84.539,Z 511.718,A -85,B 0,C 180,E1 -29516.012,E2 -29516.012} C_VEL
LIN {X 0,Y 85.076,Z 511.197,A -85,B 0,C 180,E1 -29520.003,E2 -29520.003} C_VEL
LIN {X 0,Y 84.531,Z 512.165,A -85,B 0,C 180,E1 -29524.772,E2 -29524.772} C_VEL
LIN {X 0,Y 84.159,Z 513.524,A -85,B 0,C 180,E1 -29529.617,E2 -29529.617} C_VEL
LIN {X 0,Y 83.959,Z 514.431,A -85,B 0,C 180,E1 -29532.082,E2 -29532.082} C_VEL
LIN {X 0,Y 82.821,Z 517.191,A -85,B 0,C 180,E1 -29537.51,E2 -29537.51} C_VEL
LIN {X 0,Y 82.064,Z 518.75,A -85,B 0,C 180,E1 -29540.036,E2 -29540.036} C_VEL
LIN {X 0,Y 80.076,Z 521.41,A -85,B 0,C 180,E1 -29542.849,E2 -29542.849} C_VEL
LIN {X 0,Y 76.508,Z 525.039,A -85,B 0,C 180,E1 -29546.414,E2 -29546.414} C_VEL
LIN {X 0,Y 69.107,Z 530.429,A -85,B 0,C 180,E1 -29550.567,E2 -29550.567} C_VEL
LIN {X 0,Y 61.203,Z 535.435,A -85,B 0,C 180,E1 -29556.505,E2 -29556.505} C_VEL
LIN {X 0,Y 53.91,Z 539.427,A -85,B 0,C 180,E1 -29564.193,E2 -29564.193} C_VEL
LIN {X 0,Y 47.829,Z 542.383,A -85,B 0,C 180,E1 -29574.003,E2 -29574.003} C_VEL
LIN {X 0,Y 42.62,Z 544.85,A -85,B 0,C 180,E1 -29590.744,E2 -29590.744} C_VEL
LIN {X 0,Y 41.46,Z 545.451,A -85,B 0,C 180,E1 -29600.241,E2 -29600.241} C_VEL
LIN {X 0,Y 41.326,Z 545.616,A -85,B 0,C 180,E1 -29610,E2 -29610} C_VEL
LIN {X 0,Y 41.451,Z 545.451,A -85,B 0,C 180,E1 -29619.761,E2 -29619.761} C_VEL
LIN {X 0,Y 42.615,Z 544.85,A -85,B 0,C 180,E1 -29629.258,E2 -29629.258} C_VEL
LIN {X 0,Y 47.83,Z 542.383,A -85,B 0,C 180,E1 -29645.997,E2 -29645.997} C_VEL
LIN {X 0,Y 53.913,Z 539.427,A -85,B 0,C 180,E1 -29655.803,E2 -29655.803} C_VEL
LIN {X 0,Y 61.211,Z 535.436,A -85,B 0,C 180,E1 -29663.484,E2 -29663.484} C_VEL
LIN {X 0,Y 69.009,Z 530.49,A -85,B 0,C 180,E1 -29669.385,E2 -29669.385} C_VEL
LIN {X 0,Y 76.49,Z 525.037,A -85,B 0,C 180,E1 -29673.615,E2 -29673.615} C_VEL
LIN {X 0,Y 78.917,Z 522.689,A -85,B 0,C 180,E1 -29675.896,E2 -29675.896} C_VEL
LIN {X 0,Y 81.229,Z 519.947,A -85,B 0,C 180,E1 -29678.58,E2 -29678.58} C_VEL
LIN {X 0,Y 82.151,Z 518.579,A -85,B 0,C 180,E1 -29680.225,E2 -29680.225} C_VEL
LIN {X 0,Y 83.51,Z 515.659,A -85,B 0,C 180,E1 -29685.373,E2 -29685.373} C_VEL
LIN {X 0,Y 83.961,Z 514.429,A -85,B 0,C 180,E1 -29687.918,E2 -29687.918} C_VEL
LIN {X 0,Y 84.161,Z 513.522,A -85,B 0,C 180,E1 -29690.383,E2 -29690.383} C_VEL
LIN {X 0,Y 84.593,Z 512.065,A -85,B 0,C 180,E1 -29695.516,E2 -29695.516} C_VEL
LIN {X 0,Y 85.12,Z 511.156,A -85,B 0,C 180,E1 -29699.997,E2 -29699.997} C_VEL
LIN {X 0,Y 84.141,Z 512.403,A -85,B 0,C 180,E1 -29707.384,E2 -29707.384} C_VEL
LIN {X 0,Y 83.762,Z 514.272,A -85,B 0,C 180,E1 -29714.576,E2 -29714.576} C_VEL
LIN {X 0,Y 83.345,Z 516.126,A -85,B 0,C 180,E1 -29719.709,E2 -29719.709} C_VEL
LIN {X 0,Y 82.243,Z 519.88,A -85,B 0,C 180,E1 -29726.956,E2 -29726.956} C_VEL
LIN {X 0,Y 81.355,Z 522.234,A -85,B 0,C 180,E1 -29731.217,E2 -29731.217} C_VEL
LIN {X 0,Y 79.623,Z 526.081,A -85,B 0,C 180,E1 -29737.404,E2 -29737.404} C_VEL
LIN {X 0,Y 77.503,Z 529.751,A -85,B 0,C 180,E1 -29743.496,E2 -29743.496} C_VEL
LIN {X 0,Y 75.562,Z 534.275,A -85,B 0,C 180,E1 -29752.804,E2 -29752.804} C_VEL
LIN {X 0,Y 75.98,Z 537.656,A -85,B 0,C 180,E1 -29762.453,E2 -29762.453} C_VEL
LIN {X 0,Y 77.621,Z 539.302,A -85,B 0,C 180,E1 -29768.767,E2 -29768.767} C_VEL
LIN {X 0,Y 80.327,Z 540.534,A -85,B 0,C 180,E1 -29774.783,E2 -29774.783} C_VEL
LIN {X 0,Y 85.219,Z 541.542,A -85,B 0,C 180,E1 -29781.726,E2 -29781.726} C_VEL
LIN {X 0,Y 94.393,Z 541.849,A -85,B 0,C 180,E1 -29790,E2 -29790} C_VEL
LIN {X 0,Y 85.227,Z 541.538,A -85,B 0,C 180,E1 -29798.311,E2 -29798.311} C_VEL
LIN {X 0,Y 80.208,Z 540.488,A -85,B 0,C 180,E1 -29805.466,E2 -29805.466} C_VEL
LIN {X 0,Y 76.749,Z 538.665,A -85,B 0,C 180,E1 -29813.7,E2 -29813.7} C_VEL
LIN {X 0,Y 75.459,Z 535.769,A -85,B 0,C 180,E1 -29823.052,E2 -29823.052} C_VEL
LIN {X 0,Y 75.974,Z 532.818,A -85,B 0,C 180,E1 -29830.355,E2 -29830.355} C_VEL
LIN {X 0,Y 78.37,Z 528.21,A -85,B 0,C 180,E1 -29839.023,E2 -29839.023} C_VEL
LIN {X 0,Y 80.118,Z 525.093,A -85,B 0,C 180,E1 -29844.233,E2 -29844.233} C_VEL
LIN {X 0,Y 81.226,Z 522.419,A -85,B 0,C 180,E1 -29848.536,E2 -29848.536} C_VEL
LIN {X 0,Y 81.606,Z 521.082,A -85,B 0,C 180,E1 -29851.113,E2 -29851.113} C_VEL
LIN {X 0,Y 81.249,Z 519.678,A -85,B 0,C 180,E1 -29855.154,E2 -29855.154} C_VEL
LIN {X 0,Y 80.298,Z 518.808,A -85,B 0,C 180,E1 -29859.302,E2 -29859.302} C_VEL
LIN {X 0,Y 78.481,Z 517.277,A -85,B 0,C 180,E1 -29871.209,E2 -29871.209} C_VEL
LIN {X 0,Y 78.91,Z 516.606,A -85,B 0,C 180,E1 -29874.893,E2 -29874.893} C_VEL
LIN {X 0,Y 79.672,Z 515.963,A -85,B 0,C 180,E1 -29880.003,E2 -29880.003} C_VEL
LIN {X 0,Y 79.001,Z 516.926,A -85,B 0,C 180,E1 -29885.107,E2 -29885.107} C_VEL
LIN {X 0,Y 78.447,Z 518.299,A -85,B 0,C 180,E1 -29890.325,E2 -29890.325} C_VEL
LIN {X 0,Y 77.896,Z 519.401,A -85,B 0,C 180,E1 -29893.039,E2 -29893.039} C_VEL
LIN {X 0,Y 76.527,Z 521.83,A -85,B 0,C 180,E1 -29897.635,E2 -29897.635} C_VEL
LIN {X 0,Y 73.423,Z 524.826,A -85,B 0,C 180,E1 -29901.053,E2 -29901.053} C_VEL
LIN {X 0,Y 72.069,Z 525.997,A -85,B 0,C 180,E1 -29902.12,E2 -29902.12} C_VEL
LIN {X 0,Y 63.013,Z 532.021,A -85,B 0,C 180,E1 -29906.844,E2 -29906.844} C_VEL
LIN {X 0,Y 54.456,Z 536.768,A -85,B 0,C 180,E1 -29912.98,E2 -29912.98} C_VEL
LIN {X 0,Y 46.757,Z 540.382,A -85,B 0,C 180,E1 -29921.277,E2 -29921.277} C_VEL
LIN {X 0,Y 42.263,Z 542.185,A -85,B 0,C 180,E1 -29928.306,E2 -29928.306} C_VEL
LIN {X 0,Y 35.978,Z 544.653,A -85,B 0,C 180,E1 -29947.004,E2 -29947.004} C_VEL
LIN {X 0,Y 34.48,Z 545.254,A -85,B 0,C 180,E1 -29958.239,E2 -29958.239} C_VEL
LIN {X 0,Y 34.241,Z 545.419,A -85,B 0,C 180,E1 -29970,E2 -29970} C_VEL
LIN {X 0,Y 34.473,Z 545.253,A -85,B 0,C 180,E1 -29981.763,E2 -29981.763} C_VEL
LIN {X 0,Y 35.975,Z 544.653,A -85,B 0,C 180,E1 -29992.999,E2 -29992.999} C_VEL
LIN {X 0,Y 42.263,Z 542.185,A -85,B 0,C 180,E1 -30011.694,E2 -30011.694} C_VEL
LIN {X 0,Y 49.211,Z 539.23,A -85,B 0,C 180,E1 -30021.762,E2 -30021.762} C_VEL
LIN {X 0,Y 57.264,Z 535.238,A -85,B 0,C 180,E1 -30029.214,E2 -30029.214} C_VEL
LIN {X 0,Y 66.205,Z 529.947,A -85,B 0,C 180,E1 -30035.044,E2 -30035.044} C_VEL
LIN {X 0,Y 72.046,Z 525.995,A -85,B 0,C 180,E1 -30037.924,E2 -30037.924} C_VEL
LIN {X 0,Y 74.686,Z 523.646,A -85,B 0,C 180,E1 -30040.217,E2 -30040.217} C_VEL
LIN {X 0,Y 76.546,Z 521.816,A -85,B 0,C 180,E1 -30042.37,E2 -30042.37} C_VEL
LIN {X 0,Y 77.896,Z 519.401,A -85,B 0,C 180,E1 -30046.961,E2 -30046.961} C_VEL
LIN {X 0,Y 78.481,Z 518.183,A -85,B 0,C 180,E1 -30050.074,E2 -30050.074} C_VEL
LIN {X 0,Y 79.011,Z 516.918,A -85,B 0,C 180,E1 -30054.894,E2 -30054.894} C_VEL
LIN {X 0,Y 79.713,Z 515.931,A -85,B 0,C 180,E1 -30059.997,E2 -30059.997} C_VEL
LIN {X 0,Y 78.643,Z 516.963,A -85,B 0,C 180,E1 -30067.074,E2 -30067.074} C_VEL
LIN {X 0,Y 78.351,Z 517.593,A -85,B 0,C 180,E1 -30070.332,E2 -30070.332} C_VEL
LIN {X 0,Y 77.624,Z 519.994,A -85,B 0,C 180,E1 -30078.472,E2 -30078.472} C_VEL
LIN {X 0,Y 76.653,Z 522.095,A -85,B 0,C 180,E1 -30083.533,E2 -30083.533} C_VEL
LIN {X 0,Y 75.69,Z 524.088,A -85,B 0,C 180,E1 -30087.659,E2 -30087.659} C_VEL
LIN {X 0,Y 74.521,Z 526.329,A -85,B 0,C 180,E1 -30091.923,E2 -30091.923} C_VEL
LIN {X 0,Y 73.179,Z 528.413,A -85,B 0,C 180,E1 -30095.973,E2 -30095.973} C_VEL
LIN {X 0,Y 69.927,Z 533.046,A -85,B 0,C 180,E1 -30105.29,E2 -30105.29} C_VEL
LIN {X 0,Y 68.468,Z 536.677,A -85,B 0,C 180,E1 -30115.196,E2 -30115.196} C_VEL
LIN {X 0,Y 69.638,Z 539.542,A -85,B 0,C 180,E1 -30126.192,E2 -30126.192} C_VEL
LIN {X 0,Y 75.353,Z 541.679,A -85,B 0,C 180,E1 -30139.25,E2 -30139.25} C_VEL
LIN {X 0,Y 79.772,Z 542.112,A -85,B 0,C 180,E1 -30144.946,E2 -30144.946} C_VEL
LIN {X 0,Y 85.174,Z 542.105,A -85,B 0,C 180,E1 -30150,E2 -30150} C_VEL
LIN {X 0,Y 77.928,Z 541.938,A -85,B 0,C 180,E1 -30157.256,E2 -30157.256} C_VEL
LIN {X 0,Y 71.947,Z 540.776,A -85,B 0,C 180,E1 -30167.04,E2 -30167.04} C_VEL
LIN {X 0,Y 69.467,Z 539.398,A -85,B 0,C 180,E1 -30174.429,E2 -30174.429} C_VEL
LIN {X 0,Y 68.529,Z 536.641,A -85,B 0,C 180,E1 -30184.877,E2 -30184.877} C_VEL
LIN {X 0,Y 69.956,Z 533.045,A -85,B 0,C 180,E1 -30194.686,E2 -30194.686} C_VEL
LIN {X 0,Y 72.766,Z 528.957,A -85,B 0,C 180,E1 -30203.09,E2 -30203.09} C_VEL
LIN {X 0,Y 74.898,Z 525.672,A -85,B 0,C 180,E1 -30209.399,E2 -30209.399} C_VEL
LIN {X 0,Y 76.115,Z 523.084,A -85,B 0,C 180,E1 -30214.452,E2 -30214.452} C_VEL
LIN {X 0,Y 77.018,Z 521.231,A -85,B 0,C 180,E1 -30218.595,E2 -30218.595} C_VEL
LIN {X 0,Y 77.607,Z 520.007,A -85,B 0,C 180,E1 -30221.524,E2 -30221.524} C_VEL
LIN {X 0,Y 78.35,Z 517.595,A -85,B 0,C 180,E1 -30229.668,E2 -30229.668} C_VEL
LIN {X 0,Y 78.481,Z 517.277,A -85,B 0,C 180,E1 -30231.209,E2 -30231.209} C_VEL
LIN {X 0,Y 78.178,Z 517.243,A -85,B 0,C 180,E1 -30234.049,E2 -30234.049} C_VEL
LIN {X 0,Y 77.183,Z 517.912,A -85,B 0,C 180,E1 -30236.834,E2 -30236.834} C_VEL
LIN {X 0,Y 72.983,Z 521.692,A -85,B 0,C 180,E1 -30246.47,E2 -30246.47} C_VEL
LIN {X 0,Y 72.238,Z 522.956,A -85,B 0,C 180,E1 -30251.223,E2 -30251.223} C_VEL
